LIN {X 0,Y 479.936,Z 1149.126,A -85,B 0,C 180,E1 22945.1,E2 22945.1} C_VEL
LIN {X 0,Y 479.98,Z 1146.25,A -85,B 0,C 180,E1 22942.699,E2 22942.699} C_VEL
LIN {X 0,Y 480.18,Z 1141.26,A -85,B 0,C 180,E1 22939.805,E2 22939.805} C_VEL
LIN {X 0,Y 480.58,Z 1135.396,A -85,B 0,C 180,E1 22937.259,E2 22937.259} C_VEL
LIN {X 0,Y 481.324,Z 1127.79,A -85,B 0,C 180,E1 22934.559,E2 22934.559} C_VEL
LIN {X 0,Y 482.53,Z 1118.085,A -85,B 0,C 180,E1 22931.766,E2 22931.766} C_VEL
LIN {X 0,Y 484.044,Z 1108.078,A -85,B 0,C 180,E1 22929.315,E2 22929.315} C_VEL
LIN {X 0,Y 486.397,Z 1094.541,A -85,B 0,C 180,E1 22926.496,E2 22926.496} C_VEL
LIN {X 0,Y 488.884,Z 1081.566,A -85,B 0,C 180,E1 22924.174,E2 22924.174} C_VEL
LIN {X 0,Y 492.333,Z 1064.667,A -85,B 0,C 180,E1 22921.569,E2 22921.569} C_VEL
LIN {X 0,Y 495.487,Z 1049.693,A -85,B 0,C 180,E1 22919.568,E2 22919.568} C_VEL
LIN {X 0,Y 499.695,Z 1030.069,A -85,B 0,C 180,E1 22917.298,E2 22917.298} C_VEL
LIN {X 0,Y 503.179,Z 1013.547,A -85,B 0,C 180,E1 22915.643,E2 22915.643} C_VEL
LIN {X 0,Y 507.434,Z 992.772,A -85,B 0,C 180,E1 22913.831,E2 22913.831} C_VEL
LIN {X 0,Y 511.179,Z 973.376,A -85,B 0,C 180,E1 22912.39,E2 22912.39} C_VEL
LIN {X 0,Y 515.064,Z 952.143,A -85,B 0,C 180,E1 22911.025,E2 22911.025} C_VEL
LIN {X 0,Y 518.682,Z 929.949,A -85,B 0,C 180,E1 22909.847,E2 22909.847} C_VEL
LIN {X 0,Y 521.763,Z 908.924,A -85,B 0,C 180,E1 22908.904,E2 22908.904} C_VEL
LIN {X 0,Y 524.789,Z 884.711,A -85,B 0,C 180,E1 22908.037,E2 22908.037} C_VEL
LIN {X 0,Y 526.942,Z 864.005,A -85,B 0,C 180,E1 22907.454,E2 22907.454} C_VEL
LIN {X 0,Y 528.934,Z 837.954,A -85,B 0,C 180,E1 22906.906,E2 22906.906} C_VEL
LIN {X 0,Y 532.506,Z 738.203,A -85,B 0,C 180,E1 22905.426,E2 22905.426} C_VEL
LIN {X 0,Y 540.091,Z 525.584,A -85,B 0,C 180,E1 22902.307,E2 22902.307} C_VEL
LIN {X 0,Y 527.108,Z 502.779,A -85,B 0,C 180,E1 22900.359,E2 22900.359} C_VEL
LIN {X 0,Y 515.721,Z 484.407,A -85,B 0,C 180,E1 22898.542,E2 22898.542} C_VEL
LIN {X 0,Y 504.612,Z 467.762,A -85,B 0,C 180,E1 22896.65,E2 22896.65} C_VEL
LIN {X 0,Y 495.161,Z 454.362,A -85,B 0,C 180,E1 22894.923,E2 22894.923} C_VEL
LIN {X 0,Y 490.761,Z 448.32,A -85,B 0,C 180,E1 22894.076,E2 22894.076} C_VEL
LIN {X 0,Y 486.838,Z 442.815,A -85,B 0,C 180,E1 22893.256,E2 22893.256} C_VEL
LIN {X 0,Y 485.319,Z 439.73,A -85,B 0,C 180,E1 22892.578,E2 22892.578} C_VEL
LIN {X 0,Y 483.506,Z 435.88,A -85,B 0,C 180,E1 22891.687,E2 22891.687} C_VEL
LIN {X 0,Y 482.074,Z 432.296,A -85,B 0,C 180,E1 22890.818,E2 22890.818} C_VEL
LIN {X 0,Y 482.051,Z 432.169,A -85,B 0,C 180,E1 22887.151,E2 22887.151} C_VEL
LIN {X 0,Y 482.046,Z 432.145,A -85,B 0,C 180,E1 22883.469,E2 22883.469} C_VEL
LIN {X 0,Y 482.039,Z 432.153,A -85,B 0,C 180,E1 22879.888,E2 22879.888} C_VEL
LIN {X 0,Y 482.05,Z 432.185,A -85,B 0,C 180,E1 22876.262,E2 22876.262} C_VEL
LIN {X 0,Y 482.037,Z 432.161,A -85,B 0,C 180,E1 22872.702,E2 22872.702} C_VEL
LIN {X 0,Y 482.034,Z 432.144,A -85,B 0,C 180,E1 22869.07,E2 22869.07} C_VEL
LIN {X 0,Y 482.052,Z 432.184,A -85,B 0,C 180,E1 22865.595,E2 22865.595} C_VEL
LIN {X 0,Y 482.048,Z 432.155,A -85,B 0,C 180,E1 22861.902,E2 22861.902} C_VEL
LIN {X 0,Y 482.023,Z 432.153,A -85,B 0,C 180,E1 22858.455,E2 22858.455} C_VEL
LIN {X 0,Y 482.023,Z 432.189,A -85,B 0,C 180,E1 22854.763,E2 22854.763} C_VEL
LIN {X 0,Y 482.046,Z 432.143,A -85,B 0,C 180,E1 22851.291,E2 22851.291} C_VEL
LIN {X 0,Y 482.044,Z 432.158,A -85,B 0,C 180,E1 22847.684,E2 22847.684} C_VEL
LIN {X 0,Y 482.01,Z 432.184,A -85,B 0,C 180,E1 22844.232,E2 22844.232} C_VEL
LIN {X 0,Y 482.005,Z 432.151,A -85,B 0,C 180,E1 22840.615,E2 22840.615} C_VEL
LIN {X 0,Y 482.051,Z 432.155,A -85,B 0,C 180,E1 22837.177,E2 22837.177} C_VEL
LIN {X 0,Y 482.022,Z 432.188,A -85,B 0,C 180,E1 22833.646,E2 22833.646} C_VEL
LIN {X 0,Y 481.988,Z 432.17,A -85,B 0,C 180,E1 22830.14,E2 22830.14} C_VEL
LIN {X 0,Y 482.003,Z 432.159,A -85,B 0,C 180,E1 22826.651,E2 22826.651} C_VEL
LIN {X 0,Y 482.017,Z 432.353,A -85,B 0,C 180,E1 22824.491,E2 22824.491} C_VEL
LIN {X 0,Y 482.37,Z 433.835,A -85,B 0,C 180,E1 22824.192,E2 22824.192} C_VEL
LIN {X 0,Y 484.285,Z 436.852,A -85,B 0,C 180,E1 22823.771,E2 22823.771} C_VEL
LIN {X 0,Y 486.647,Z 438.772,A -85,B 0,C 180,E1 22823.317,E2 22823.317} C_VEL
LIN {X 0,Y 489.004,Z 442.512,A -85,B 0,C 180,E1 22822.827,E2 22822.827} C_VEL
LIN {X 0,Y 491.314,Z 444.857,A -85,B 0,C 180,E1 22822.39,E2 22822.39} C_VEL
LIN {X 0,Y 494.506,Z 449.067,A -85,B 0,C 180,E1 22821.776,E2 22821.776} C_VEL
LIN {X 0,Y 496.224,Z 451.276,A -85,B 0,C 180,E1 22821.454,E2 22821.454} C_VEL
LIN {X 0,Y 503.923,Z 461.08,A -85,B 0,C 180,E1 22820.067,E2 22820.067} C_VEL
LIN {X 0,Y 515.356,Z 476.674,A -85,B 0,C 180,E1 22818.131,E2 22818.131} C_VEL
LIN {X 0,Y 527.952,Z 494.875,A -85,B 0,C 180,E1 22816.156,E2 22816.156} C_VEL
LIN {X 0,Y 540.315,Z 514.018,A -85,B 0,C 180,E1 22814.349,E2 22814.349} C_VEL
LIN {X 0,Y 531.611,Z 754.844,A -85,B 0,C 180,E1 22810.823,E2 22810.823} C_VEL
LIN {X 0,Y 529.419,Z 812.429,A -85,B 0,C 180,E1 22809.954,E2 22809.954} C_VEL
LIN {X 0,Y 527.614,Z 836.833,A -85,B 0,C 180,E1 22809.41,E2 22809.41} C_VEL
LIN {X 0,Y 525.485,Z 858.718,A -85,B 0,C 180,E1 22808.766,E2 22808.766} C_VEL
LIN {X 0,Y 522.555,Z 882.977,A -85,B 0,C 180,E1 22807.847,E2 22807.847} C_VEL
LIN {X 0,Y 519.79,Z 902.352,A -85,B 0,C 180,E1 22806.952,E2 22806.952} C_VEL
LIN {X 0,Y 516.232,Z 924.536,A -85,B 0,C 180,E1 22805.738,E2 22805.738} C_VEL
LIN {X 0,Y 512.66,Z 944.242,A -85,B 0,C 180,E1 22804.445,E2 22804.445} C_VEL
LIN {X 0,Y 509.031,Z 962.981,A -85,B 0,C 180,E1 22803.031,E2 22803.031} C_VEL
LIN {X 0,Y 504.72,Z 983.574,A -85,B 0,C 180,E1 22801.214,E2 22801.214} C_VEL
LIN {X 0,Y 501.128,Z 1000.134,A -85,B 0,C 180,E1 22799.527,E2 22799.527} C_VEL
LIN {X 0,Y 499.238,Z 1008.711,A -85,B 0,C 180,E1 22798.556,E2 22798.556} C_VEL
LIN {X 0,Y 497.144,Z 1014.273,A -85,B 0,C 180,E1 22797.965,E2 22797.965} C_VEL
LIN {X 0,Y 488.33,Z 1028.661,A -85,B 0,C 180,E1 22796.469,E2 22796.469} C_VEL
LIN {X 0,Y 486.663,Z 1032.843,A -85,B 0,C 180,E1 22795.904,E2 22795.904} C_VEL
LIN {X 0,Y 483.204,Z 1047.996,A -85,B 0,C 180,E1 22793.539,E2 22793.539} C_VEL
LIN {X 0,Y 480.254,Z 1061.231,A -85,B 0,C 180,E1 22791.112,E2 22791.112} C_VEL
LIN {X 0,Y 477.712,Z 1073.52,A -85,B 0,C 180,E1 22788.527,E2 22788.527} C_VEL
LIN {X 0,Y 475.693,Z 1084.165,A -85,B 0,C 180,E1 22785.858,E2 22785.858} C_VEL
LIN {X 0,Y 474.325,Z 1092.525,A -85,B 0,C 180,E1 22783.408,E2 22783.408} C_VEL
LIN {X 0,Y 473.141,Z 1101.135,A -85,B 0,C 180,E1 22780.348,E2 22780.348} C_VEL
LIN {X 0,Y 472.538,Z 1106.877,A -85,B 0,C 180,E1 22777.783,E2 22777.783} C_VEL
LIN {X 0,Y 472.182,Z 1111.811,A -85,B 0,C 180,E1 22774.981,E2 22774.981} C_VEL
LIN {X 0,Y 472.022,Z 1115.222,A -85,B 0,C 180,E1 22772.064,E2 22772.064} C_VEL
LIN {X 0,Y 471.975,Z 1117.08,A -85,B 0,C 180,E1 22769.42,E2 22769.42} C_VEL
LIN {X 0,Y 471.949,Z 1117.65,A -85,B 0,C 180,E1 22766.477,E2 22766.477} C_VEL
LIN {X 0,Y 471.985,Z 1116.842,A -85,B 0,C 180,E1 22763.92,E2 22763.92} C_VEL
LIN {X 0,Y 472.055,Z 1114.793,A -85,B 0,C 180,E1 22761.228,E2 22761.228} C_VEL
LIN {X 0,Y 472.266,Z 1110.779,A -85,B 0,C 180,E1 22758.149,E2 22758.149} C_VEL
LIN {X 0,Y 472.687,Z 1106.041,A -85,B 0,C 180,E1 22755.546,E2 22755.546} C_VEL
LIN {X 0,Y 473.537,Z 1099.04,A -85,B 0,C 180,E1 22752.552,E2 22752.552} C_VEL
LIN {X 0,Y 474.692,Z 1091.317,A -85,B 0,C 180,E1 22749.919,E2 22749.919} C_VEL
LIN {X 0,Y 476.475,Z 1081.561,A -85,B 0,C 180,E1 22747.11,E2 22747.11} C_VEL
LIN {X 0,Y 478.802,Z 1070.113,A -85,B 0,C 180,E1 22744.387,E2 22744.387} C_VEL
LIN {X 0,Y 481.716,Z 1057.311,A -85,B 0,C 180,E1 22741.754,E2 22741.754} C_VEL
LIN {X 0,Y 485.097,Z 1042.937,A -85,B 0,C 180,E1 22739.257,E2 22739.257} C_VEL
LIN {X 0,Y 488.946,Z 1027.419,A -85,B 0,C 180,E1 22736.906,E2 22736.906} C_VEL
LIN {X 0,Y 493.024,Z 1010.801,A -85,B 0,C 180,E1 22734.761,E2 22734.761} C_VEL
LIN {X 0,Y 496.931,Z 994.799,A -85,B 0,C 180,E1 22732.946,E2 22732.946} C_VEL
LIN {X 0,Y 501.49,Z 975.341,A -85,B 0,C 180,E1 22731.042,E2 22731.042} C_VEL
LIN {X 0,Y 505.451,Z 957.608,A -85,B 0,C 180,E1 22729.544,E2 22729.544} C_VEL
LIN {X 0,Y 510.033,Z 935.666,A -85,B 0,C 180,E1 22727.954,E2 22727.954} C_VEL
LIN {X 0,Y 513.708,Z 916.026,A -85,B 0,C 180,E1 22726.753,E2 22726.753} C_VEL
LIN {X 0,Y 517.485,Z 894.109,A -85,B 0,C 180,E1 22725.616,E2 22725.616} C_VEL
LIN {X 0,Y 520.64,Z 871.877,A -85,B 0,C 180,E1 22724.678,E2 22724.678} C_VEL
LIN {X 0,Y 523.211,Z 850.767,A -85,B 0,C 180,E1 22723.951,E2 22723.951} C_VEL
LIN {X 0,Y 525.614,Z 825.467,A -85,B 0,C 180,E1 22723.286,E2 22723.286} C_VEL
LIN {X 0,Y 527.005,Z 803.925,A -85,B 0,C 180,E1 22722.873,E2 22722.873} C_VEL
LIN {X 0,Y 537.124,Z 553.916,A -85,B 0,C 180,E1 22719.149,E2 22719.149} C_VEL
LIN {X 0,Y 538.478,Z 519.428,A -85,B 0,C 180,E1 22718.621,E2 22718.621} C_VEL
LIN {X 0,Y 526.57,Z 501.373,A -85,B 0,C 180,E1 22716.67,E2 22716.67} C_VEL
LIN {X 0,Y 513.397,Z 482.898,A -85,B 0,C 180,E1 22714.328,E2 22714.328} C_VEL
LIN {X 0,Y 502.204,Z 468.261,A -85,B 0,C 180,E1 22712.147,E2 22712.147} C_VEL
LIN {X 0,Y 496.887,Z 461.776,A -85,B 0,C 180,E1 22711.041,E2 22711.041} C_VEL
LIN {X 0,Y 492.914,Z 456.709,A -85,B 0,C 180,E1 22710.17,E2 22710.17} C_VEL
LIN {X 0,Y 489.386,Z 452.141,A -85,B 0,C 180,E1 22709.364,E2 22709.364} C_VEL
LIN {X 0,Y 485.532,Z 448.038,A -85,B 0,C 180,E1 22708.473,E2 22708.473} C_VEL
LIN {X 0,Y 484.051,Z 445.687,A -85,B 0,C 180,E1 22708.098,E2 22708.098} C_VEL
LIN {X 0,Y 480.94,Z 442.93,A -85,B 0,C 180,E1 22707.353,E2 22707.353} C_VEL
LIN {X 0,Y 478.923,Z 439.552,A -85,B 0,C 180,E1 22706.806,E2 22706.806} C_VEL
LIN {X 0,Y 475.792,Z 437.238,A -85,B 0,C 180,E1 22706.021,E2 22706.021} C_VEL
LIN {X 0,Y 474.203,Z 433.97,A -85,B 0,C 180,E1 22705.477,E2 22705.477} C_VEL
LIN {X 0,Y 474.091,Z 433.21,A -85,B 0,C 180,E1 22705.083,E2 22705.083} C_VEL
LIN {X 0,Y 474.059,Z 433.17,A -85,B 0,C 180,E1 22701.661,E2 22701.661} C_VEL
LIN {X 0,Y 474.081,Z 433.179,A -85,B 0,C 180,E1 22698.062,E2 22698.062} C_VEL
LIN {X 0,Y 474.123,Z 433.153,A -85,B 0,C 180,E1 22694.533,E2 22694.533} C_VEL
LIN {X 0,Y 474.093,Z 433.142,A -85,B 0,C 180,E1 22690.942,E2 22690.942} C_VEL
LIN {X 0,Y 474.072,Z 433.146,A -85,B 0,C 180,E1 22687.392,E2 22687.392} C_VEL
LIN {X 0,Y 474.087,Z 433.165,A -85,B 0,C 180,E1 22683.749,E2 22683.749} C_VEL
LIN {X 0,Y 474.121,Z 433.16,A -85,B 0,C 180,E1 22680.121,E2 22680.121} C_VEL
LIN {X 0,Y 474.106,Z 433.137,A -85,B 0,C 180,E1 22676.494,E2 22676.494} C_VEL
LIN {X 0,Y 474.1,Z 433.137,A -85,B 0,C 180,E1 22672.852,E2 22672.852} C_VEL
LIN {X 0,Y 474.095,Z 433.156,A -85,B 0,C 180,E1 22669.181,E2 22669.181} C_VEL
LIN {X 0,Y 474.108,Z 433.175,A -85,B 0,C 180,E1 22665.465,E2 22665.465} C_VEL
LIN {X 0,Y 474.109,Z 433.157,A -85,B 0,C 180,E1 22661.812,E2 22661.812} C_VEL
LIN {X 0,Y 474.095,Z 433.122,A -85,B 0,C 180,E1 22658.123,E2 22658.123} C_VEL
LIN {X 0,Y 474.105,Z 433.14,A -85,B 0,C 180,E1 22654.51,E2 22654.51} C_VEL
LIN {X 0,Y 474.169,Z 433.53,A -85,B 0,C 180,E1 22653.136,E2 22653.136} C_VEL
LIN {X 0,Y 475.766,Z 437.121,A -85,B 0,C 180,E1 22652.052,E2 22652.052} C_VEL
LIN {X 0,Y 476.842,Z 439.144,A -85,B 0,C 180,E1 22651.439,E2 22651.439} C_VEL
LIN {X 0,Y 478.321,Z 441.84,A -85,B 0,C 180,E1 22650.749,E2 22650.749} C_VEL
LIN {X 0,Y 480.674,Z 444.989,A -85,B 0,C 180,E1 22650.119,E2 22650.119} C_VEL
LIN {X 0,Y 484.461,Z 449.557,A -85,B 0,C 180,E1 22649.178,E2 22649.178} C_VEL
LIN {X 0,Y 493.093,Z 461.044,A -85,B 0,C 180,E1 22647.15,E2 22647.15} C_VEL
LIN {X 0,Y 496.711,Z 465.928,A -85,B 0,C 180,E1 22646.352,E2 22646.352} C_VEL
LIN {X 0,Y 505.532,Z 478.146,A -85,B 0,C 180,E1 22644.513,E2 22644.513} C_VEL
LIN {X 0,Y 517.369,Z 495.765,A -85,B 0,C 180,E1 22642.236,E2 22642.236} C_VEL
LIN {X 0,Y 529.249,Z 514.827,A -85,B 0,C 180,E1 22640.138,E2 22640.138} C_VEL
LIN {X 0,Y 538.374,Z 530.866,A -85,B 0,C 180,E1 22638.624,E2 22638.624} C_VEL
LIN {X 0,Y 529.453,Z 752.304,A -85,B 0,C 180,E1 22635.324,E2 22635.324} C_VEL
LIN {X 0,Y 525.979,Z 837.792,A -85,B 0,C 180,E1 22634.032,E2 22634.032} C_VEL
LIN {X 0,Y 523.839,Z 863.39,A -85,B 0,C 180,E1 22633.489,E2 22633.489} C_VEL
LIN {X 0,Y 521.554,Z 883.538,A -85,B 0,C 180,E1 22632.923,E2 22632.923} C_VEL
LIN {X 0,Y 518.464,Z 906.572,A -85,B 0,C 180,E1 22632.109,E2 22632.109} C_VEL
LIN {X 0,Y 515.038,Z 927.934,A -85,B 0,C 180,E1 22631.158,E2 22631.158} C_VEL
LIN {X 0,Y 511.484,Z 947.966,A -85,B 0,C 180,E1 22630.101,E2 22630.101} C_VEL
LIN {X 0,Y 506.92,Z 971.138,A -85,B 0,C 180,E1 22628.638,E2 22628.638} C_VEL
LIN {X 0,Y 502.967,Z 989.767,A -85,B 0,C 180,E1 22627.254,E2 22627.254} C_VEL
LIN {X 0,Y 498.144,Z 1011.239,A -85,B 0,C 180,E1 22625.394,E2 22625.394} C_VEL
LIN {X 0,Y 494.168,Z 1028.309,A -85,B 0,C 180,E1 22623.67,E2 22623.67} C_VEL
LIN {X 0,Y 490.033,Z 1046.043,A -85,B 0,C 180,E1 22621.628,E2 22621.628} C_VEL
LIN {X 0,Y 486.163,Z 1062.323,A -85,B 0,C 180,E1 22619.443,E2 22619.443} C_VEL
LIN {X 0,Y 482.714,Z 1077.589,A -85,B 0,C 180,E1 22617.111,E2 22617.111} C_VEL
LIN {X 0,Y 479.55,Z 1092.099,A -85,B 0,C 180,E1 22614.515,E2 22614.515} C_VEL
LIN {X 0,Y 477.183,Z 1104.197,A -85,B 0,C 180,E1 22612.029,E2 22612.029} C_VEL
LIN {X 0,Y 475.106,Z 1116.023,A -85,B 0,C 180,E1 22609.166,E2 22609.166} C_VEL
LIN {X 0,Y 473.768,Z 1125.193,A -85,B 0,C 180,E1 22606.554,E2 22606.554} C_VEL
LIN {X 0,Y 472.752,Z 1134.133,A -85,B 0,C 180,E1 22603.453,E2 22603.453} C_VEL
LIN {X 0,Y 472.266,Z 1140.124,A -85,B 0,C 180,E1 22600.861,E2 22600.861} C_VEL
LIN {X 0,Y 471.998,Z 1145.405,A -85,B 0,C 180,E1 22597.915,E2 22597.915} C_VEL
LIN {X 0,Y 471.932,Z 1148.649,A -85,B 0,C 180,E1 22595.252,E2 22595.252} C_VEL
LIN {X 0,Y 471.932,Z 1150.44,A -85,B 0,C 180,E1 22592.915,E2 22592.915} C_VEL
LIN {X 0,Y 471.949,Z 1151.281,A -85,B 0,C 180,E1 22590.243,E2 22590.243} C_VEL
LIN {X 0,Y 471.94,Z 1150.604,A -85,B 0,C 180,E1 22587.45,E2 22587.45} C_VEL
LIN {X 0,Y 471.937,Z 1148.827,A -85,B 0,C 180,E1 22585.017,E2 22585.017} C_VEL
LIN {X 0,Y 471.98,Z 1145.943,A -85,B 0,C 180,E1 22582.575,E2 22582.575} C_VEL
LIN {X 0,Y 472.199,Z 1140.94,A -85,B 0,C 180,E1 22579.631,E2 22579.631} C_VEL
LIN {X 0,Y 472.625,Z 1135.067,A -85,B 0,C 180,E1 22577.041,E2 22577.041} C_VEL
LIN {X 0,Y 473.411,Z 1127.509,A -85,B 0,C 180,E1 22574.315,E2 22574.315} C_VEL
LIN {X 0,Y 474.701,Z 1117.728,A -85,B 0,C 180,E1 22571.454,E2 22571.454} C_VEL
LIN {X 0,Y 476.296,Z 1107.71,A -85,B 0,C 180,E1 22568.962,E2 22568.962} C_VEL
LIN {X 0,Y 478.782,Z 1094.151,A -85,B 0,C 180,E1 22566.099,E2 22566.099} C_VEL
LIN {X 0,Y 481.301,Z 1081.658,A -85,B 0,C 180,E1 22563.828,E2 22563.828} C_VEL
LIN {X 0,Y 484.946,Z 1064.601,A -85,B 0,C 180,E1 22561.153,E2 22561.153} C_VEL
LIN {X 0,Y 488.302,Z 1049.388,A -85,B 0,C 180,E1 22559.091,E2 22559.091} C_VEL
LIN {X 0,Y 492.724,Z 1029.594,A -85,B 0,C 180,E1 22556.776,E2 22556.776} C_VEL
LIN {X 0,Y 496.453,Z 1012.59,A -85,B 0,C 180,E1 22555.058,E2 22555.058} C_VEL
LIN {X 0,Y 501.127,Z 990.544,A -85,B 0,C 180,E1 22553.141,E2 22553.141} C_VEL
LIN {X 0,Y 504.863,Z 971.911,A -85,B 0,C 180,E1 22551.756,E2 22551.756} C_VEL
LIN {X 0,Y 509.062,Z 949.487,A -85,B 0,C 180,E1 22550.33,E2 22550.33} C_VEL
LIN {X 0,Y 512.46,Z 929.277,A -85,B 0,C 180,E1 22549.257,E2 22549.257} C_VEL
LIN {X 0,Y 515.769,Z 907.446,A -85,B 0,C 180,E1 22548.278,E2 22548.278} C_VEL
LIN {X 0,Y 518.777,Z 883.834,A -85,B 0,C 180,E1 22547.437,E2 22547.437} C_VEL
LIN {X 0,Y 520.974,Z 863.298,A -85,B 0,C 180,E1 22546.859,E2 22546.859} C_VEL
LIN {X 0,Y 523.033,Z 836.601,A -85,B 0,C 180,E1 22546.3,E2 22546.3} C_VEL
LIN {X 0,Y 530.859,Z 624.102,A -85,B 0,C 180,E1 22543.147,E2 22543.147} C_VEL
LIN {X 0,Y 534.336,Z 528.71,A -85,B 0,C 180,E1 22541.719,E2 22541.719} C_VEL
LIN {X 0,Y 521.84,Z 506.736,A -85,B 0,C 180,E1 22539.79,E2 22539.79} C_VEL
LIN {X 0,Y 509.772,Z 487.18,A -85,B 0,C 180,E1 22537.803,E2 22537.803} C_VEL
LIN {X 0,Y 497.334,Z 468.611,A -85,B 0,C 180,E1 22535.594,E2 22535.594} C_VEL
LIN {X 0,Y 487.735,Z 455.202,A -85,B 0,C 180,E1 22533.75,E2 22533.75} C_VEL
LIN {X 0,Y 481.103,Z 446.349,A -85,B 0,C 180,E1 22532.391,E2 22532.391} C_VEL
LIN {X 0,Y 478.14,Z 441.839,A -85,B 0,C 180,E1 22531.661,E2 22531.661} C_VEL
LIN {X 0,Y 475.595,Z 436.916,A -85,B 0,C 180,E1 22530.443,E2 22530.443} C_VEL
LIN {X 0,Y 474.129,Z 433.295,A -85,B 0,C 180,E1 22529.5,E2 22529.5} C_VEL
LIN {X 0,Y 474.098,Z 433.161,A -85,B 0,C 180,E1 22525.885,E2 22525.885} C_VEL
LIN {X 0,Y 474.102,Z 433.162,A -85,B 0,C 180,E1 22522.18,E2 22522.18} C_VEL
LIN {X 0,Y 474.106,Z 433.137,A -85,B 0,C 180,E1 22518.57,E2 22518.57} C_VEL
LIN {X 0,Y 474.1,Z 433.139,A -85,B 0,C 180,E1 22514.91,E2 22514.91} C_VEL
LIN {X 0,Y 474.108,Z 433.175,A -85,B 0,C 180,E1 22511.279,E2 22511.279} C_VEL
LIN {X 0,Y 474.11,Z 433.139,A -85,B 0,C 180,E1 22507.595,E2 22507.595} C_VEL
LIN {X 0,Y 474.105,Z 433.136,A -85,B 0,C 180,E1 22503.991,E2 22503.991} C_VEL
LIN {X 0,Y 474.092,Z 433.176,A -85,B 0,C 180,E1 22500.363,E2 22500.363} C_VEL
LIN {X 0,Y 474.081,Z 433.136,A -85,B 0,C 180,E1 22496.735,E2 22496.735} C_VEL
LIN {X 0,Y 474.11,Z 433.144,A -85,B 0,C 180,E1 22493.217,E2 22493.217} C_VEL
LIN {X 0,Y 474.113,Z 433.169,A -85,B 0,C 180,E1 22489.55,E2 22489.55} C_VEL
LIN {X 0,Y 474.081,Z 433.133,A -85,B 0,C 180,E1 22485.963,E2 22485.963} C_VEL
LIN {X 0,Y 474.067,Z 433.155,A -85,B 0,C 180,E1 22482.43,E2 22482.43} C_VEL
LIN {X 0,Y 474.084,Z 433.172,A -85,B 0,C 180,E1 22478.859,E2 22478.859} C_VEL
LIN {X 0,Y 474.104,Z 433.136,A -85,B 0,C 180,E1 22475.366,E2 22475.366} C_VEL
LIN {X 0,Y 474.064,Z 433.143,A -85,B 0,C 180,E1 22471.806,E2 22471.806} C_VEL
LIN {X 0,Y 474.048,Z 433.159,A -85,B 0,C 180,E1 22468.216,E2 22468.216} C_VEL
LIN {X 0,Y 474.06,Z 433.271,A -85,B 0,C 180,E1 22465.944,E2 22465.944} C_VEL
LIN {X 0,Y 474.423,Z 434.745,A -85,B 0,C 180,E1 22465.624,E2 22465.624} C_VEL
LIN {X 0,Y 476.306,Z 437.77,A -85,B 0,C 180,E1 22465.18,E2 22465.18} C_VEL
LIN {X 0,Y 478.828,Z 439.895,A -85,B 0,C 180,E1 22464.659,E2 22464.659} C_VEL
LIN {X 0,Y 481.264,Z 443.655,A -85,B 0,C 180,E1 22464.123,E2 22464.123} C_VEL
LIN {X 0,Y 483.6,Z 445.904,A -85,B 0,C 180,E1 22463.656,E2 22463.656} C_VEL
LIN {X 0,Y 486.679,Z 450.083,A -85,B 0,C 180,E1 22463.025,E2 22463.025} C_VEL
LIN {X 0,Y 488.487,Z 452.236,A -85,B 0,C 180,E1 22462.67,E2 22462.67} C_VEL
LIN {X 0,Y 493.304,Z 458.45,A -85,B 0,C 180,E1 22461.74,E2 22461.74} C_VEL
LIN {X 0,Y 500.474,Z 467.61,A -85,B 0,C 180,E1 22460.426,E2 22460.426} C_VEL
LIN {X 0,Y 511.731,Z 483.101,A -85,B 0,C 180,E1 22458.48,E2 22458.48} C_VEL
LIN {X 0,Y 524.073,Z 501.11,A -85,B 0,C 180,E1 22456.505,E2 22456.505} C_VEL
LIN {X 0,Y 534.671,Z 517.793,A -85,B 0,C 180,E1 22454.915,E2 22454.915} C_VEL
LIN {X 0,Y 525.544,Z 760.909,A -85,B 0,C 180,E1 22451.329,E2 22451.329} C_VEL
LIN {X 0,Y 523.446,Z 813.486,A -85,B 0,C 180,E1 22450.524,E2 22450.524} C_VEL
LIN {X 0,Y 521.571,Z 837.655,A -85,B 0,C 180,E1 22449.976,E2 22449.976} C_VEL
LIN {X 0,Y 519.314,Z 860.093,A -85,B 0,C 180,E1 22449.306,E2 22449.306} C_VEL
LIN {X 0,Y 516.425,Z 883.033,A -85,B 0,C 180,E1 22448.427,E2 22448.427} C_VEL
LIN {X 0,Y 513.451,Z 903.213,A -85,B 0,C 180,E1 22447.486,E2 22447.486} C_VEL
LIN {X 0,Y 509.588,Z 926.256,A -85,B 0,C 180,E1 22446.2,E2 22446.2} C_VEL
LIN {X 0,Y 505.899,Z 945.877,A -85,B 0,C 180,E1 22444.891,E2 22444.891} C_VEL
LIN {X 0,Y 501.75,Z 966.474,A -85,B 0,C 180,E1 22443.3,E2 22443.3} C_VEL
LIN {X 0,Y 497.537,Z 985.58,A -85,B 0,C 180,E1 22441.558,E2 22441.558} C_VEL
LIN {X 0,Y 493.351,Z 1004.247,A -85,B 0,C 180,E1 22439.603,E2 22439.603} C_VEL
LIN {X 0,Y 489.356,Z 1021.307,A -85,B 0,C 180,E1 22437.502,E2 22437.502} C_VEL
LIN {X 0,Y 486.663,Z 1032.843,A -85,B 0,C 180,E1 22435.904,E2 22435.904} C_VEL
LIN {X 0,Y 484.627,Z 1037.843,A -85,B 0,C 180,E1 22435.234,E2 22435.234} C_VEL
LIN {X 0,Y 476.305,Z 1049.996,A -85,B 0,C 180,E1 22433.6,E2 22433.6} C_VEL
LIN {X 0,Y 474.375,Z 1054.367,A -85,B 0,C 180,E1 22432.87,E2 22432.87} C_VEL
LIN {X 0,Y 471.109,Z 1068.831,A -85,B 0,C 180,E1 22429.981,E2 22429.981} C_VEL
LIN {X 0,Y 468.907,Z 1079.415,A -85,B 0,C 180,E1 22427.498,E2 22427.498} C_VEL
LIN {X 0,Y 466.861,Z 1090.562,A -85,B 0,C 180,E1 22424.385,E2 22424.385} C_VEL
LIN {X 0,Y 465.647,Z 1098.464,A -85,B 0,C 180,E1 22421.712,E2 22421.712} C_VEL
LIN {X 0,Y 464.717,Z 1105.998,A -85,B 0,C 180,E1 22418.538,E2 22418.538} C_VEL
LIN {X 0,Y 464.28,Z 1110.751,A -85,B 0,C 180,E1 22415.934,E2 22415.934} C_VEL
LIN {X 0,Y 464.063,Z 1114.639,A -85,B 0,C 180,E1 22413.088,E2 22413.088} C_VEL
LIN {X 0,Y 464.005,Z 1116.998,A -85,B 0,C 180,E1 22410.123,E2 22410.123} C_VEL
LIN {X 0,Y 463.958,Z 1117.893,A -85,B 0,C 180,E1 22407.53,E2 22407.53} C_VEL
LIN {X 0,Y 463.979,Z 1117.439,A -85,B 0,C 180,E1 22404.435,E2 22404.435} C_VEL
LIN {X 0,Y 464.047,Z 1115.6,A -85,B 0,C 180,E1 22401.699,E2 22401.699} C_VEL
LIN {X 0,Y 464.22,Z 1112.369,A -85,B 0,C 180,E1 22398.822,E2 22398.822} C_VEL
LIN {X 0,Y 464.655,Z 1107.257,A -85,B 0,C 180,E1 22395.799,E2 22395.799} C_VEL
LIN {X 0,Y 465.357,Z 1101.455,A -85,B 0,C 180,E1 22393.138,E2 22393.138} C_VEL
LIN {X 0,Y 466.722,Z 1092.696,A -85,B 0,C 180,E1 22389.954,E2 22389.954} C_VEL
LIN {X 0,Y 468.316,Z 1084.161,A -85,B 0,C 180,E1 22387.399,E2 22387.399} C_VEL
LIN {X 0,Y 470.925,Z 1071.955,A -85,B 0,C 180,E1 22384.333,E2 22384.333} C_VEL
LIN {X 0,Y 473.577,Z 1060.588,A -85,B 0,C 180,E1 22381.911,E2 22381.911} C_VEL
LIN {X 0,Y 477.265,Z 1045.788,A -85,B 0,C 180,E1 22379.201,E2 22379.201} C_VEL
LIN {X 0,Y 480.854,Z 1031.702,A -85,B 0,C 180,E1 22376.989,E2 22376.989} C_VEL
LIN {X 0,Y 485.368,Z 1014.37,A -85,B 0,C 180,E1 22374.628,E2 22374.628} C_VEL
LIN {X 0,Y 489.446,Z 998.29,A -85,B 0,C 180,E1 22372.746,E2 22372.746} C_VEL
LIN {X 0,Y 494.075,Z 979.746,A -85,B 0,C 180,E1 22370.845,E2 22370.845} C_VEL
LIN {X 0,Y 498.541,Z 960.464,A -85,B 0,C 180,E1 22369.168,E2 22369.168} C_VEL
LIN {X 0,Y 502.778,Z 941.198,A -85,B 0,C 180,E1 22367.715,E2 22367.715} C_VEL
LIN {X 0,Y 507.119,Z 919.301,A -85,B 0,C 180,E1 22366.32,E2 22366.32} C_VEL
LIN {X 0,Y 510.741,Z 899.097,A -85,B 0,C 180,E1 22365.238,E2 22365.238} C_VEL
LIN {X 0,Y 514.539,Z 874.389,A -85,B 0,C 180,E1 22364.147,E2 22364.147} C_VEL
LIN {X 0,Y 517.198,Z 853.451,A -85,B 0,C 180,E1 22363.407,E2 22363.407} C_VEL
LIN {X 0,Y 519.756,Z 828.599,A -85,B 0,C 180,E1 22362.725,E2 22362.725} C_VEL
LIN {X 0,Y 521.316,Z 805.933,A -85,B 0,C 180,E1 22362.277,E2 22362.277} C_VEL
LIN {X 0,Y 531.53,Z 563.128,A -85,B 0,C 180,E1 22358.631,E2 22358.631} C_VEL
LIN {X 0,Y 533.235,Z 523.387,A -85,B 0,C 180,E1 22358.03,E2 22358.03} C_VEL
LIN {X 0,Y 521.943,Z 506.222,A -85,B 0,C 180,E1 22356.126,E2 22356.126} C_VEL
LIN {X 0,Y 509.696,Z 488.932,A -85,B 0,C 180,E1 22353.892,E2 22353.892} C_VEL
LIN {X 0,Y 499.038,Z 474.875,A -85,B 0,C 180,E1 22351.766,E2 22351.766} C_VEL
LIN {X 0,Y 493.434,Z 467.961,A -85,B 0,C 180,E1 22350.572,E2 22350.572} C_VEL
LIN {X 0,Y 489.86,Z 463.368,A -85,B 0,C 180,E1 22349.77,E2 22349.77} C_VEL
LIN {X 0,Y 485.917,Z 458.419,A -85,B 0,C 180,E1 22348.852,E2 22348.852} C_VEL
LIN {X 0,Y 482.383,Z 454.261,A -85,B 0,C 180,E1 22348.002,E2 22348.002} C_VEL
LIN {X 0,Y 481.32,Z 452.783,A -85,B 0,C 180,E1 22347.732,E2 22347.732} C_VEL
LIN {X 0,Y 477.967,Z 449.361,A -85,B 0,C 180,E1 22346.897,E2 22346.897} C_VEL
LIN {X 0,Y 476.25,Z 446.767,A -85,B 0,C 180,E1 22346.43,E2 22346.43} C_VEL
LIN {X 0,Y 473.103,Z 443.984,A -85,B 0,C 180,E1 22345.608,E2 22345.608} C_VEL
LIN {X 0,Y 471.223,Z 440.672,A -85,B 0,C 180,E1 22345.045,E2 22345.045} C_VEL
LIN {X 0,Y 467.883,Z 438.226,A -85,B 0,C 180,E1 22344.124,E2 22344.124} C_VEL
LIN {X 0,Y 466.263,Z 434.951,A -85,B 0,C 180,E1 22343.508,E2 22343.508} C_VEL
LIN {X 0,Y 466.159,Z 434.177,A -85,B 0,C 180,E1 22342.978,E2 22342.978} C_VEL
LIN {X 0,Y 466.126,Z 434.139,A -85,B 0,C 180,E1 22339.42,E2 22339.42} C_VEL
LIN {X 0,Y 466.128,Z 434.133,A -85,B 0,C 180,E1 22335.809,E2 22335.809} C_VEL
LIN {X 0,Y 466.162,Z 434.134,A -85,B 0,C 180,E1 22332.26,E2 22332.26} C_VEL
LIN {X 0,Y 466.178,Z 434.155,A -85,B 0,C 180,E1 22328.587,E2 22328.587} C_VEL
LIN {X 0,Y 466.158,Z 434.156,A -85,B 0,C 180,E1 22324.922,E2 22324.922} C_VEL
LIN {X 0,Y 466.144,Z 434.129,A -85,B 0,C 180,E1 22321.229,E2 22321.229} C_VEL
LIN {X 0,Y 466.148,Z 434.123,A -85,B 0,C 180,E1 22317.541,E2 22317.541} C_VEL
LIN {X 0,Y 466.17,Z 434.138,A -85,B 0,C 180,E1 22313.843,E2 22313.843} C_VEL
LIN {X 0,Y 466.173,Z 434.162,A -85,B 0,C 180,E1 22310.12,E2 22310.12} C_VEL
LIN {X 0,Y 466.168,Z 434.143,A -85,B 0,C 180,E1 22306.353,E2 22306.353} C_VEL
LIN {X 0,Y 466.164,Z 434.13,A -85,B 0,C 180,E1 22302.782,E2 22302.782} C_VEL
LIN {X 0,Y 466.164,Z 434.115,A -85,B 0,C 180,E1 22299.142,E2 22299.142} C_VEL
LIN {X 0,Y 466.172,Z 434.16,A -85,B 0,C 180,E1 22295.546,E2 22295.546} C_VEL
LIN {X 0,Y 466.25,Z 434.646,A -85,B 0,C 180,E1 22294.873,E2 22294.873} C_VEL
LIN {X 0,Y 467.82,Z 438.088,A -85,B 0,C 180,E1 22293.741,E2 22293.741} C_VEL
LIN {X 0,Y 468.97,Z 440.146,A -85,B 0,C 180,E1 22293.059,E2 22293.059} C_VEL
LIN {X 0,Y 472.33,Z 444.518,A -85,B 0,C 180,E1 22292.037,E2 22292.037} C_VEL
LIN {X 0,Y 477.82,Z 451.575,A -85,B 0,C 180,E1 22290.543,E2 22290.543} C_VEL
LIN {X 0,Y 481.863,Z 456.649,A -85,B 0,C 180,E1 22289.512,E2 22289.512} C_VEL
LIN {X 0,Y 489.945,Z 467.466,A -85,B 0,C 180,E1 22287.573,E2 22287.573} C_VEL
LIN {X 0,Y 497.176,Z 477.385,A -85,B 0,C 180,E1 22285.968,E2 22285.968} C_VEL
LIN {X 0,Y 506.9,Z 491.496,A -85,B 0,C 180,E1 22283.962,E2 22283.962} C_VEL
LIN {X 0,Y 518.453,Z 509.357,A -85,B 0,C 180,E1 22281.768,E2 22281.768} C_VEL
LIN {X 0,Y 530.467,Z 529.55,A -85,B 0,C 180,E1 22279.666,E2 22279.666} C_VEL
LIN {X 0,Y 533.048,Z 534.482,A -85,B 0,C 180,E1 22279.227,E2 22279.227} C_VEL
LIN {X 0,Y 523.844,Z 754.793,A -85,B 0,C 180,E1 22275.921,E2 22275.921} C_VEL
LIN {X 0,Y 520.347,Z 837.619,A -85,B 0,C 180,E1 22274.659,E2 22274.659} C_VEL
LIN {X 0,Y 518.135,Z 863.216,A -85,B 0,C 180,E1 22274.112,E2 22274.112} C_VEL
LIN {X 0,Y 515.763,Z 883.49,A -85,B 0,C 180,E1 22273.54,E2 22273.54} C_VEL
LIN {X 0,Y 512.506,Z 906.844,A -85,B 0,C 180,E1 22272.707,E2 22272.707} C_VEL
LIN {X 0,Y 508.987,Z 928.03,A -85,B 0,C 180,E1 22271.756,E2 22271.756} C_VEL
LIN {X 0,Y 505.13,Z 949.022,A -85,B 0,C 180,E1 22270.636,E2 22270.636} C_VEL
LIN {X 0,Y 500.55,Z 971.289,A -85,B 0,C 180,E1 22269.208,E2 22269.208} C_VEL
LIN {X 0,Y 496.49,Z 989.723,A -85,B 0,C 180,E1 22267.824,E2 22267.824} C_VEL
LIN {X 0,Y 491.398,Z 1011.451,A -85,B 0,C 180,E1 22265.919,E2 22265.919} C_VEL
LIN {X 0,Y 487.193,Z 1028.757,A -85,B 0,C 180,E1 22264.147,E2 22264.147} C_VEL
LIN {X 0,Y 482.529,Z 1047.763,A -85,B 0,C 180,E1 22261.898,E2 22261.898} C_VEL
LIN {X 0,Y 478.762,Z 1063.016,A -85,B 0,C 180,E1 22259.806,E2 22259.806} C_VEL
LIN {X 0,Y 475,Z 1078.882,A -85,B 0,C 180,E1 22257.316,E2 22257.316} C_VEL
LIN {X 0,Y 471.88,Z 1092.545,A -85,B 0,C 180,E1 22254.806,E2 22254.806} C_VEL
LIN {X 0,Y 469.303,Z 1105.147,A -85,B 0,C 180,E1 22252.155,E2 22252.155} C_VEL
LIN {X 0,Y 467.237,Z 1116.263,A -85,B 0,C 180,E1 22249.372,E2 22249.372} C_VEL
LIN {X 0,Y 465.84,Z 1125.37,A -85,B 0,C 180,E1 22246.716,E2 22246.716} C_VEL
LIN {X 0,Y 464.81,Z 1133.884,A -85,B 0,C 180,E1 22243.688,E2 22243.688} C_VEL
LIN {X 0,Y 464.289,Z 1139.869,A -85,B 0,C 180,E1 22241.05,E2 22241.05} C_VEL
LIN {X 0,Y 464.007,Z 1145.138,A -85,B 0,C 180,E1 22238.052,E2 22238.052} C_VEL
LIN {X 0,Y 463.938,Z 1148.283,A -85,B 0,C 180,E1 22235.442,E2 22235.442} C_VEL
LIN {X 0,Y 463.939,Z 1150.093,A -85,B 0,C 180,E1 22233.089,E2 22233.089} C_VEL
LIN {X 0,Y 463.947,Z 1150.929,A -85,B 0,C 180,E1 22230.617,E2 22230.617} C_VEL
LIN {X 0,Y 463.953,Z 1150.449,A -85,B 0,C 180,E1 22227.653,E2 22227.653} C_VEL
LIN {X 0,Y 463.941,Z 1148.644,A -85,B 0,C 180,E1 22225.054,E2 22225.054} C_VEL
LIN {X 0,Y 463.983,Z 1145.965,A -85,B 0,C 180,E1 22222.695,E2 22222.695} C_VEL
LIN {X 0,Y 464.176,Z 1141.395,A -85,B 0,C 180,E1 22219.826,E2 22219.826} C_VEL
LIN {X 0,Y 464.647,Z 1135.047,A -85,B 0,C 180,E1 22216.941,E2 22216.941} C_VEL
LIN {X 0,Y 465.434,Z 1127.757,A -85,B 0,C 180,E1 22214.247,E2 22214.247} C_VEL
LIN {X 0,Y 466.841,Z 1117.646,A -85,B 0,C 180,E1 22211.207,E2 22211.207} C_VEL
LIN {X 0,Y 468.472,Z 1107.865,A -85,B 0,C 180,E1 22208.725,E2 22208.725} C_VEL
LIN {X 0,Y 471.064,Z 1094.407,A -85,B 0,C 180,E1 22205.816,E2 22205.816} C_VEL
LIN {X 0,Y 473.684,Z 1081.976,A -85,B 0,C 180,E1 22203.511,E2 22203.511} C_VEL
LIN {X 0,Y 477.103,Z 1066.757,A -85,B 0,C 180,E1 22201.045,E2 22201.045} C_VEL
LIN {X 0,Y 480.767,Z 1050.692,A -85,B 0,C 180,E1 22198.811,E2 22198.811} C_VEL
LIN {X 0,Y 484.923,Z 1033.073,A -85,B 0,C 180,E1 22196.666,E2 22196.666} C_VEL
LIN {X 0,Y 489.155,Z 1014.413,A -85,B 0,C 180,E1 22194.727,E2 22194.727} C_VEL
LIN {X 0,Y 493.504,Z 994.998,A -85,B 0,C 180,E1 22192.967,E2 22192.967} C_VEL
LIN {X 0,Y 497.899,Z 973.893,A -85,B 0,C 180,E1 22191.35,E2 22191.35} C_VEL
LIN {X 0,Y 502.052,Z 952.797,A -85,B 0,C 180,E1 22189.962,E2 22189.962} C_VEL
LIN {X 0,Y 505.914,Z 930.892,A -85,B 0,C 180,E1 22188.766,E2 22188.766} C_VEL
LIN {X 0,Y 508.983,Z 911.37,A -85,B 0,C 180,E1 22187.865,E2 22187.865} C_VEL
LIN {X 0,Y 512.411,Z 886.458,A -85,B 0,C 180,E1 22186.933,E2 22186.933} C_VEL
LIN {X 0,Y 514.793,Z 865.163,A -85,B 0,C 180,E1 22186.316,E2 22186.316} C_VEL
LIN {X 0,Y 516.918,Z 840.547,A -85,B 0,C 180,E1 22185.77,E2 22185.77} C_VEL
LIN {X 0,Y 519.086,Z 787.879,A -85,B 0,C 180,E1 22184.96,E2 22184.96} C_VEL
LIN {X 0,Y 527.339,Z 570.067,A -85,B 0,C 180,E1 22181.714,E2 22181.714} C_VEL
LIN {X 0,Y 528.751,Z 532.081,A -85,B 0,C 180,E1 22181.136,E2 22181.136} C_VEL
LIN {X 0,Y 516.831,Z 511.042,A -85,B 0,C 180,E1 22179.245,E2 22179.245} C_VEL
LIN {X 0,Y 505.116,Z 492.034,A -85,B 0,C 180,E1 22177.264,E2 22177.264} C_VEL
LIN {X 0,Y 493.184,Z 474.029,A -85,B 0,C 180,E1 22175.084,E2 22175.084} C_VEL
LIN {X 0,Y 482.355,Z 458.77,A -85,B 0,C 180,E1 22172.931,E2 22172.931} C_VEL
LIN {X 0,Y 474.196,Z 447.898,A -85,B 0,C 180,E1 22171.176,E2 22171.176} C_VEL
LIN {X 0,Y 469.517,Z 441.736,A -85,B 0,C 180,E1 22170.066,E2 22170.066} C_VEL
LIN {X 0,Y 467.824,Z 438.092,A -85,B 0,C 180,E1 22169.164,E2 22169.164} C_VEL
LIN {X 0,Y 466.181,Z 434.331,A -85,B 0,C 180,E1 22168.113,E2 22168.113} C_VEL
LIN {X 0,Y 466.165,Z 434.12,A -85,B 0,C 180,E1 22164.455,E2 22164.455} C_VEL
LIN {X 0,Y 466.166,Z 434.149,A -85,B 0,C 180,E1 22160.858,E2 22160.858} C_VEL
LIN {X 0,Y 466.169,Z 434.154,A -85,B 0,C 180,E1 22157.217,E2 22157.217} C_VEL
LIN {X 0,Y 466.168,Z 434.121,A -85,B 0,C 180,E1 22153.521,E2 22153.521} C_VEL
LIN {X 0,Y 466.167,Z 434.13,A -85,B 0,C 180,E1 22149.881,E2 22149.881} C_VEL
LIN {X 0,Y 466.174,Z 434.161,A -85,B 0,C 180,E1 22146.157,E2 22146.157} C_VEL
LIN {X 0,Y 466.149,Z 434.123,A -85,B 0,C 180,E1 22142.459,E2 22142.459} C_VEL
LIN {X 0,Y 466.147,Z 434.134,A -85,B 0,C 180,E1 22138.771,E2 22138.771} C_VEL
LIN {X 0,Y 466.159,Z 434.16,A -85,B 0,C 180,E1 22135.078,E2 22135.078} C_VEL
LIN {X 0,Y 466.173,Z 434.116,A -85,B 0,C 180,E1 22131.489,E2 22131.489} C_VEL
LIN {X 0,Y 466.155,Z 434.139,A -85,B 0,C 180,E1 22127.865,E2 22127.865} C_VEL
LIN {X 0,Y 466.131,Z 434.156,A -85,B 0,C 180,E1 22124.319,E2 22124.319} C_VEL
LIN {X 0,Y 466.132,Z 434.125,A -85,B 0,C 180,E1 22120.707,E2 22120.707} C_VEL
LIN {X 0,Y 466.171,Z 434.13,A -85,B 0,C 180,E1 22117.156,E2 22117.156} C_VEL
LIN {X 0,Y 466.159,Z 434.161,A -85,B 0,C 180,E1 22113.438,E2 22113.438} C_VEL
LIN {X 0,Y 466.113,Z 434.148,A -85,B 0,C 180,E1 22110.011,E2 22110.011} C_VEL
LIN {X 0,Y 466.18,Z 434.399,A -85,B 0,C 180,E1 22107.428,E2 22107.428} C_VEL
LIN {X 0,Y 466.621,Z 435.984,A -85,B 0,C 180,E1 22107.122,E2 22107.122} C_VEL
LIN {X 0,Y 468.47,Z 438.866,A -85,B 0,C 180,E1 22106.66,E2 22106.66} C_VEL
LIN {X 0,Y 470.989,Z 440.815,A -85,B 0,C 180,E1 22106.107,E2 22106.107} C_VEL
LIN {X 0,Y 473.323,Z 444.536,A -85,B 0,C 180,E1 22105.554,E2 22105.554} C_VEL
LIN {X 0,Y 475.912,Z 447.08,A -85,B 0,C 180,E1 22105,E2 22105} C_VEL
LIN {X 0,Y 478.945,Z 451.16,A -85,B 0,C 180,E1 22104.339,E2 22104.339} C_VEL
LIN {X 0,Y 480.708,Z 453.074,A -85,B 0,C 180,E1 22103.975,E2 22103.975} C_VEL
LIN {X 0,Y 484.363,Z 457.611,A -85,B 0,C 180,E1 22103.226,E2 22103.226} C_VEL
LIN {X 0,Y 496.977,Z 474.031,A -85,B 0,C 180,E1 22100.802,E2 22100.802} C_VEL
LIN {X 0,Y 508.335,Z 489.827,A -85,B 0,C 180,E1 22098.799,E2 22098.799} C_VEL
LIN {X 0,Y 520.431,Z 507.672,A -85,B 0,C 180,E1 22096.826,E2 22096.826} C_VEL
LIN {X 0,Y 529.075,Z 521.491,A -85,B 0,C 180,E1 22095.494,E2 22095.494} C_VEL
LIN {X 0,Y 519.585,Z 765.228,A -85,B 0,C 180,E1 22091.872,E2 22091.872} C_VEL
LIN {X 0,Y 517.533,Z 814.324,A -85,B 0,C 180,E1 22091.111,E2 22091.111} C_VEL
LIN {X 0,Y 515.591,Z 838.342,A -85,B 0,C 180,E1 22090.558,E2 22090.558} C_VEL
LIN {X 0,Y 513.2,Z 861.35,A -85,B 0,C 180,E1 22089.863,E2 22089.863} C_VEL
LIN {X 0,Y 510.223,Z 883.965,A -85,B 0,C 180,E1 22088.982,E2 22088.982} C_VEL
LIN {X 0,Y 507.157,Z 904.07,A -85,B 0,C 180,E1 22088.033,E2 22088.033} C_VEL
LIN {X 0,Y 502.994,Z 927.883,A -85,B 0,C 180,E1 22086.681,E2 22086.681} C_VEL
LIN {X 0,Y 499.345,Z 946.615,A -85,B 0,C 180,E1 22085.414,E2 22085.414} C_VEL
LIN {X 0,Y 495.059,Z 967.104,A -85,B 0,C 180,E1 22083.81,E2 22083.81} C_VEL
LIN {X 0,Y 490.862,Z 985.491,A -85,B 0,C 180,E1 22082.118,E2 22082.118} C_VEL
LIN {X 0,Y 486.662,Z 1003.468,A -85,B 0,C 180,E1 22080.224,E2 22080.224} C_VEL
LIN {X 0,Y 482.41,Z 1020.936,A -85,B 0,C 180,E1 22078.067,E2 22078.067} C_VEL
LIN {X 0,Y 478.877,Z 1035.531,A -85,B 0,C 180,E1 22076.007,E2 22076.007} C_VEL
LIN {X 0,Y 475.076,Z 1051.339,A -85,B 0,C 180,E1 22073.415,E2 22073.415} C_VEL
LIN {X 0,Y 474.375,Z 1054.367,A -85,B 0,C 180,E1 22072.87,E2 22072.87} C_VEL
LIN {X 0,Y 472.478,Z 1058.695,A -85,B 0,C 180,E1 22072.122,E2 22072.122} C_VEL
LIN {X 0,Y 464.443,Z 1069.275,A -85,B 0,C 180,E1 22070.269,E2 22070.269} C_VEL
LIN {X 0,Y 462.655,Z 1073.083,A -85,B 0,C 180,E1 22069.465,E2 22069.465} C_VEL
LIN {X 0,Y 460.238,Z 1084.547,A -85,B 0,C 180,E1 22066.535,E2 22066.535} C_VEL
LIN {X 0,Y 458.691,Z 1092.931,A -85,B 0,C 180,E1 22064.003,E2 22064.003} C_VEL
LIN {X 0,Y 457.35,Z 1101.583,A -85,B 0,C 180,E1 22060.837,E2 22060.837} C_VEL
LIN {X 0,Y 456.661,Z 1107.344,A -85,B 0,C 180,E1 22058.182,E2 22058.182} C_VEL
LIN {X 0,Y 456.222,Z 1112.482,A -85,B 0,C 180,E1 22055.156,E2 22055.156} C_VEL
LIN {X 0,Y 456.043,Z 1115.745,A -85,B 0,C 180,E1 22052.262,E2 22052.262} C_VEL
LIN {X 0,Y 455.99,Z 1117.569,A -85,B 0,C 180,E1 22049.623,E2 22049.623} C_VEL
LIN {X 0,Y 455.96,Z 1118.228,A -85,B 0,C 180,E1 22046.48,E2 22046.48} C_VEL
LIN {X 0,Y 456,Z 1117.44,A -85,B 0,C 180,E1 22043.832,E2 22043.832} C_VEL
LIN {X 0,Y 456.075,Z 1115.524,A -85,B 0,C 180,E1 22041.172,E2 22041.172} C_VEL
LIN {X 0,Y 456.316,Z 1111.644,A -85,B 0,C 180,E1 22037.985,E2 22037.985} C_VEL
LIN {X 0,Y 456.788,Z 1106.977,A -85,B 0,C 180,E1 22035.29,E2 22035.29} C_VEL
LIN {X 0,Y 457.72,Z 1100.301,A -85,B 0,C 180,E1 22032.26,E2 22032.26} C_VEL
LIN {X 0,Y 459.105,Z 1092.076,A -85,B 0,C 180,E1 22029.34,E2 22029.34} C_VEL
LIN {X 0,Y 461.059,Z 1082.513,A -85,B 0,C 180,E1 22026.482,E2 22026.482} C_VEL
LIN {X 0,Y 463.688,Z 1070.954,A -85,B 0,C 180,E1 22023.627,E2 22023.627} C_VEL
LIN {X 0,Y 466.749,Z 1058.817,A -85,B 0,C 180,E1 22021.043,E2 22021.043} C_VEL
LIN {X 0,Y 470.467,Z 1044.537,A -85,B 0,C 180,E1 22018.458,E2 22018.458} C_VEL
LIN {X 0,Y 474.125,Z 1030.926,A -85,B 0,C 180,E1 22016.313,E2 22016.313} C_VEL
LIN {X 0,Y 478.948,Z 1013.119,A -85,B 0,C 180,E1 22013.895,E2 22013.895} C_VEL
LIN {X 0,Y 483.103,Z 997.408,A -85,B 0,C 180,E1 22012.052,E2 22012.052} C_VEL
LIN {X 0,Y 487.998,Z 978.366,A -85,B 0,C 180,E1 22010.109,E2 22010.109} C_VEL
LIN {X 0,Y 492.507,Z 959.637,A -85,B 0,C 180,E1 22008.481,E2 22008.481} C_VEL
LIN {X 0,Y 497.187,Z 939.124,A -85,B 0,C 180,E1 22006.939,E2 22006.939} C_VEL
LIN {X 0,Y 501.324,Z 918.603,A -85,B 0,C 180,E1 22005.647,E2 22005.647} C_VEL
LIN {X 0,Y 504.904,Z 899.228,A -85,B 0,C 180,E1 22004.607,E2 22004.607} C_VEL
LIN {X 0,Y 508.799,Z 874.67,A -85,B 0,C 180,E1 22003.518,E2 22003.518} C_VEL
LIN {X 0,Y 511.528,Z 853.844,A -85,B 0,C 180,E1 22002.777,E2 22002.777} C_VEL
LIN {X 0,Y 514.155,Z 829.146,A -85,B 0,C 180,E1 22002.095,E2 22002.095} C_VEL
LIN {X 0,Y 515.778,Z 806.329,A -85,B 0,C 180,E1 22001.64,E2 22001.64} C_VEL
LIN {X 0,Y 526.332,Z 564.5,A -85,B 0,C 180,E1 21997.984,E2 21997.984} C_VEL
LIN {X 0,Y 527.938,Z 527.132,A -85,B 0,C 180,E1 21997.408,E2 21997.408} C_VEL
LIN {X 0,Y 516.313,Z 509.543,A -85,B 0,C 180,E1 21995.383,E2 21995.383} C_VEL
LIN {X 0,Y 504.067,Z 492.174,A -85,B 0,C 180,E1 21993.059,E2 21993.059} C_VEL
LIN {X 0,Y 494.815,Z 480.196,A -85,B 0,C 180,E1 21991.152,E2 21991.152} C_VEL
LIN {X 0,Y 487.178,Z 470.373,A -85,B 0,C 180,E1 21989.443,E2 21989.443} C_VEL
LIN {X 0,Y 483.049,Z 465.259,A -85,B 0,C 180,E1 21988.464,E2 21988.464} C_VEL
LIN {X 0,Y 479.372,Z 460.643,A -85,B 0,C 180,E1 21987.551,E2 21987.551} C_VEL
LIN {X 0,Y 475.126,Z 455.924,A -85,B 0,C 180,E1 21986.463,E2 21986.463} C_VEL
LIN {X 0,Y 473.822,Z 454.049,A -85,B 0,C 180,E1 21986.103,E2 21986.103} C_VEL
LIN {X 0,Y 470.538,Z 450.851,A -85,B 0,C 180,E1 21985.218,E2 21985.218} C_VEL
LIN {X 0,Y 468.647,Z 447.92,A -85,B 0,C 180,E1 21984.653,E2 21984.653} C_VEL
LIN {X 0,Y 465.399,Z 445.12,A -85,B 0,C 180,E1 21983.722,E2 21983.722} C_VEL
LIN {X 0,Y 463.375,Z 441.7,A -85,B 0,C 180,E1 21983.057,E2 21983.057} C_VEL
LIN {X 0,Y 459.996,Z 439.306,A -85,B 0,C 180,E1 21982.022,E2 21982.022} C_VEL
LIN {X 0,Y 458.325,Z 435.914,A -85,B 0,C 180,E1 21981.321,E2 21981.321} C_VEL
LIN {X 0,Y 458.23,Z 435.149,A -85,B 0,C 180,E1 21980.835,E2 21980.835} C_VEL
LIN {X 0,Y 458.196,Z 435.138,A -85,B 0,C 180,E1 21977.265,E2 21977.265} C_VEL
LIN {X 0,Y 458.193,Z 435.158,A -85,B 0,C 180,E1 21973.632,E2 21973.632} C_VEL
LIN {X 0,Y 458.208,Z 435.136,A -85,B 0,C 180,E1 21969.927,E2 21969.927} C_VEL
LIN {X 0,Y 458.235,Z 435.115,A -85,B 0,C 180,E1 21966.264,E2 21966.264} C_VEL
LIN {X 0,Y 458.226,Z 435.114,A -85,B 0,C 180,E1 21962.626,E2 21962.626} C_VEL
LIN {X 0,Y 458.216,Z 435.138,A -85,B 0,C 180,E1 21959,E2 21959} C_VEL
LIN {X 0,Y 458.214,Z 435.142,A -85,B 0,C 180,E1 21955.243,E2 21955.243} C_VEL
LIN {X 0,Y 458.218,Z 435.12,A -85,B 0,C 180,E1 21951.467,E2 21951.467} C_VEL
LIN {X 0,Y 458.229,Z 435.113,A -85,B 0,C 180,E1 21947.78,E2 21947.78} C_VEL
LIN {X 0,Y 458.226,Z 435.124,A -85,B 0,C 180,E1 21944.171,E2 21944.171} C_VEL
LIN {X 0,Y 458.23,Z 435.138,A -85,B 0,C 180,E1 21940.497,E2 21940.497} C_VEL
LIN {X 0,Y 458.259,Z 435.333,A -85,B 0,C 180,E1 21936.976,E2 21936.976} C_VEL
LIN {X 0,Y 459.864,Z 439.085,A -85,B 0,C 180,E1 21935.599,E2 21935.599} C_VEL
LIN {X 0,Y 461.538,Z 441.272,A -85,B 0,C 180,E1 21934.942,E2 21934.942} C_VEL
LIN {X 0,Y 464.807,Z 445.386,A -85,B 0,C 180,E1 21933.901,E2 21933.901} C_VEL
LIN {X 0,Y 466.789,Z 447.737,A -85,B 0,C 180,E1 21933.301,E2 21933.301} C_VEL
LIN {X 0,Y 474.993,Z 458.16,A -85,B 0,C 180,E1 21930.973,E2 21930.973} C_VEL
LIN {X 0,Y 479.492,Z 464.038,A -85,B 0,C 180,E1 21929.796,E2 21929.796} C_VEL
LIN {X 0,Y 486.602,Z 473.556,A -85,B 0,C 180,E1 21928.054,E2 21928.054} C_VEL
LIN {X 0,Y 494.644,Z 484.816,A -85,B 0,C 180,E1 21926.227,E2 21926.227} C_VEL
LIN {X 0,Y 503.803,Z 498.27,A -85,B 0,C 180,E1 21924.303,E2 21924.303} C_VEL
LIN {X 0,Y 515.039,Z 515.905,A -85,B 0,C 180,E1 21922.123,E2 21922.123} C_VEL
LIN {X 0,Y 526.653,Z 535.696,A -85,B 0,C 180,E1 21920.044,E2 21920.044} C_VEL
LIN {X 0,Y 527.784,Z 538.067,A -85,B 0,C 180,E1 21919.842,E2 21919.842} C_VEL
LIN {X 0,Y 518.3,Z 757.174,A -85,B 0,C 180,E1 21916.533,E2 21916.533} C_VEL
LIN {X 0,Y 514.776,Z 837.46,A -85,B 0,C 180,E1 21915.299,E2 21915.299} C_VEL
LIN {X 0,Y 512.508,Z 862.949,A -85,B 0,C 180,E1 21914.752,E2 21914.752} C_VEL
LIN {X 0,Y 510.058,Z 883.242,A -85,B 0,C 180,E1 21914.178,E2 21914.178} C_VEL
LIN {X 0,Y 506.563,Z 907.36,A -85,B 0,C 180,E1 21913.308,E2 21913.308} C_VEL
LIN {X 0,Y 502.993,Z 928.132,A -85,B 0,C 180,E1 21912.368,E2 21912.368} C_VEL
LIN {X 0,Y 499.011,Z 949.079,A -85,B 0,C 180,E1 21911.242,E2 21911.242} C_VEL
LIN {X 0,Y 494.287,Z 971.195,A -85,B 0,C 180,E1 21909.81,E2 21909.81} C_VEL
LIN {X 0,Y 490.109,Z 989.487,A -85,B 0,C 180,E1 21908.425,E2 21908.425} C_VEL
LIN {X 0,Y 484.837,Z 1011.123,A -85,B 0,C 180,E1 21906.511,E2 21906.511} C_VEL
LIN {X 0,Y 480.535,Z 1028.092,A -85,B 0,C 180,E1 21904.76,E2 21904.76} C_VEL
LIN {X 0,Y 475.775,Z 1046.69,A -85,B 0,C 180,E1 21902.548,E2 21902.548} C_VEL
LIN {X 0,Y 471.728,Z 1062.357,A -85,B 0,C 180,E1 21900.38,E2 21900.38} C_VEL
LIN {X 0,Y 467.827,Z 1077.992,A -85,B 0,C 180,E1 21897.909,E2 21897.909} C_VEL
LIN {X 0,Y 464.421,Z 1092.143,A -85,B 0,C 180,E1 21895.276,E2 21895.276} C_VEL
LIN {X 0,Y 461.646,Z 1104.937,A -85,B 0,C 180,E1 21892.543,E2 21892.543} C_VEL
LIN {X 0,Y 459.453,Z 1116.038,A -85,B 0,C 180,E1 21889.714,E2 21889.714} C_VEL
LIN {X 0,Y 457.966,Z 1125.173,A -85,B 0,C 180,E1 21887,E2 21887} C_VEL
LIN {X 0,Y 456.869,Z 1133.636,A -85,B 0,C 180,E1 21883.93,E2 21883.93} C_VEL
LIN {X 0,Y 456.328,Z 1139.354,A -85,B 0,C 180,E1 21881.374,E2 21881.374} C_VEL
LIN {X 0,Y 456.048,Z 1144.538,A -85,B 0,C 180,E1 21878.447,E2 21878.447} C_VEL
LIN {X 0,Y 455.944,Z 1148.012,A -85,B 0,C 180,E1 21875.537,E2 21875.537} C_VEL
LIN {X 0,Y 455.945,Z 1149.817,A -85,B 0,C 180,E1 21873.143,E2 21873.143} C_VEL
LIN {X 0,Y 455.952,Z 1150.647,A -85,B 0,C 180,E1 21870.628,E2 21870.628} C_VEL
LIN {X 0,Y 455.956,Z 1150.156,A -85,B 0,C 180,E1 21867.612,E2 21867.612} C_VEL
LIN {X 0,Y 455.942,Z 1148.343,A -85,B 0,C 180,E1 21864.967,E2 21864.967} C_VEL
LIN {X 0,Y 455.983,Z 1145.656,A -85,B 0,C 180,E1 21862.566,E2 21862.566} C_VEL
LIN {X 0,Y 456.195,Z 1141.074,A -85,B 0,C 180,E1 21859.646,E2 21859.646} C_VEL
LIN {X 0,Y 456.699,Z 1134.713,A -85,B 0,C 180,E1 21856.71,E2 21856.71} C_VEL
LIN {X 0,Y 457.519,Z 1127.549,A -85,B 0,C 180,E1 21854.016,E2 21854.016} C_VEL
LIN {X 0,Y 459.002,Z 1117.475,A -85,B 0,C 180,E1 21850.928,E2 21850.928} C_VEL
LIN {X 0,Y 460.761,Z 1107.492,A -85,B 0,C 180,E1 21848.351,E2 21848.351} C_VEL
LIN {X 0,Y 463.492,Z 1094.011,A -85,B 0,C 180,E1 21845.395,E2 21845.395} C_VEL
LIN {X 0,Y 466.198,Z 1081.781,A -85,B 0,C 180,E1 21843.093,E2 21843.093} C_VEL
LIN {X 0,Y 469.829,Z 1066.323,A -85,B 0,C 180,E1 21840.553,E2 21840.553} C_VEL
LIN {X 0,Y 473.558,Z 1050.716,A -85,B 0,C 180,E1 21838.352,E2 21838.352} C_VEL
LIN {X 0,Y 477.917,Z 1032.969,A -85,B 0,C 180,E1 21836.161,E2 21836.161} C_VEL
LIN {X 0,Y 482.263,Z 1014.532,A -85,B 0,C 180,E1 21834.219,E2 21834.219} C_VEL
LIN {X 0,Y 486.694,Z 995.475,A -85,B 0,C 180,E1 21832.469,E2 21832.469} C_VEL
LIN {X 0,Y 491.308,Z 974.228,A -85,B 0,C 180,E1 21830.816,E2 21830.816} C_VEL
LIN {X 0,Y 495.23,Z 954.933,A -85,B 0,C 180,E1 21829.524,E2 21829.524} C_VEL
LIN {X 0,Y 499.599,Z 931.356,A -85,B 0,C 180,E1 21828.205,E2 21828.205} C_VEL
LIN {X 0,Y 502.762,Z 911.935,A -85,B 0,C 180,E1 21827.298,E2 21827.298} C_VEL
LIN {X 0,Y 506.204,Z 888.088,A -85,B 0,C 180,E1 21826.385,E2 21826.385} C_VEL
LIN {X 0,Y 508.796,Z 865.728,A -85,B 0,C 180,E1 21825.727,E2 21825.727} C_VEL
LIN {X 0,Y 510.94,Z 842.046,A -85,B 0,C 180,E1 21825.19,E2 21825.19} C_VEL
LIN {X 0,Y 512.735,Z 802.682,A -85,B 0,C 180,E1 21824.564,E2 21824.564} C_VEL
LIN {X 0,Y 521.304,Z 584.245,A -85,B 0,C 180,E1 21821.286,E2 21821.286} C_VEL
LIN {X 0,Y 523.225,Z 535.391,A -85,B 0,C 180,E1 21820.541,E2 21820.541} C_VEL
LIN {X 0,Y 510.89,Z 513.738,A -85,B 0,C 180,E1 21818.526,E2 21818.526} C_VEL
LIN {X 0,Y 499.443,Z 495.113,A -85,B 0,C 180,E1 21816.52,E2 21816.52} C_VEL
LIN {X 0,Y 487.656,Z 477.463,A -85,B 0,C 180,E1 21814.288,E2 21814.288} C_VEL
LIN {X 0,Y 478.544,Z 464.563,A -85,B 0,C 180,E1 21812.415,E2 21812.415} C_VEL
LIN {X 0,Y 471.078,Z 454.5,A -85,B 0,C 180,E1 21810.766,E2 21810.766} C_VEL
LIN {X 0,Y 463.622,Z 444.759,A -85,B 0,C 180,E1 21808.994,E2 21808.994} C_VEL
LIN {X 0,Y 460.864,Z 440.923,A -85,B 0,C 180,E1 21808.228,E2 21808.228} C_VEL
LIN {X 0,Y 458.404,Z 436.061,A -85,B 0,C 180,E1 21806.841,E2 21806.841} C_VEL
LIN {X 0,Y 458.246,Z 435.248,A -85,B 0,C 180,E1 21806.54,E2 21806.54} C_VEL
LIN {X 0,Y 458.23,Z 435.118,A -85,B 0,C 180,E1 21802.856,E2 21802.856} C_VEL
LIN {X 0,Y 458.226,Z 435.11,A -85,B 0,C 180,E1 21799.106,E2 21799.106} C_VEL
LIN {X 0,Y 458.236,Z 435.123,A -85,B 0,C 180,E1 21795.439,E2 21795.439} C_VEL
LIN {X 0,Y 458.231,Z 435.15,A -85,B 0,C 180,E1 21791.709,E2 21791.709} C_VEL
LIN {X 0,Y 458.231,Z 435.109,A -85,B 0,C 180,E1 21787.901,E2 21787.901} C_VEL
LIN {X 0,Y 458.221,Z 435.116,A -85,B 0,C 180,E1 21784.255,E2 21784.255} C_VEL
LIN {X 0,Y 458.211,Z 435.154,A -85,B 0,C 180,E1 21780.625,E2 21780.625} C_VEL
LIN {X 0,Y 458.212,Z 435.107,A -85,B 0,C 180,E1 21776.998,E2 21776.998} C_VEL
LIN {X 0,Y 458.241,Z 435.121,A -85,B 0,C 180,E1 21773.359,E2 21773.359} C_VEL
LIN {X 0,Y 458.235,Z 435.147,A -85,B 0,C 180,E1 21769.565,E2 21769.565} C_VEL
LIN {X 0,Y 458.202,Z 435.109,A -85,B 0,C 180,E1 21765.982,E2 21765.982} C_VEL
LIN {X 0,Y 458.189,Z 435.127,A -85,B 0,C 180,E1 21762.342,E2 21762.342} C_VEL
LIN {X 0,Y 458.193,Z 435.156,A -85,B 0,C 180,E1 21758.627,E2 21758.627} C_VEL
LIN {X 0,Y 458.222,Z 435.117,A -85,B 0,C 180,E1 21755.093,E2 21755.093} C_VEL
LIN {X 0,Y 458.213,Z 435.114,A -85,B 0,C 180,E1 21751.452,E2 21751.452} C_VEL
LIN {X 0,Y 458.258,Z 435.307,A -85,B 0,C 180,E1 21749.152,E2 21749.152} C_VEL
LIN {X 0,Y 458.552,Z 436.683,A -85,B 0,C 180,E1 21748.828,E2 21748.828} C_VEL
LIN {X 0,Y 460.249,Z 439.592,A -85,B 0,C 180,E1 21748.355,E2 21748.355} C_VEL
LIN {X 0,Y 463.267,Z 441.929,A -85,B 0,C 180,E1 21747.638,E2 21747.638} C_VEL
LIN {X 0,Y 465.567,Z 445.648,A -85,B 0,C 180,E1 21747.05,E2 21747.05} C_VEL
LIN {X 0,Y 468.238,Z 448.147,A -85,B 0,C 180,E1 21746.44,E2 21746.44} C_VEL
LIN {X 0,Y 471.326,Z 452.319,A -85,B 0,C 180,E1 21745.719,E2 21745.719} C_VEL
LIN {X 0,Y 473.144,Z 454.307,A -85,B 0,C 180,E1 21745.319,E2 21745.319} C_VEL
LIN {X 0,Y 476.798,Z 458.787,A -85,B 0,C 180,E1 21744.523,E2 21744.523} C_VEL
LIN {X 0,Y 486.739,Z 471.628,A -85,B 0,C 180,E1 21742.476,E2 21742.476} C_VEL
LIN {X 0,Y 494.491,Z 481.892,A -85,B 0,C 180,E1 21740.996,E2 21740.996} C_VEL
LIN {X 0,Y 504.679,Z 496.145,A -85,B 0,C 180,E1 21739.17,E2 21739.17} C_VEL
LIN {X 0,Y 516.647,Z 513.988,A -85,B 0,C 180,E1 21737.176,E2 21737.176} C_VEL
LIN {X 0,Y 523.532,Z 525.25,A -85,B 0,C 180,E1 21736.084,E2 21736.084} C_VEL
LIN {X 0,Y 513.666,Z 769.671,A -85,B 0,C 180,E1 21732.426,E2 21732.426} C_VEL
LIN {X 0,Y 511.677,Z 815.015,A -85,B 0,C 180,E1 21731.713,E2 21731.713} C_VEL
LIN {X 0,Y 509.68,Z 838.855,A -85,B 0,C 180,E1 21731.158,E2 21731.158} C_VEL
LIN {X 0,Y 507.174,Z 862.22,A -85,B 0,C 180,E1 21730.445,E2 21730.445} C_VEL
LIN {X 0,Y 504.07,Z 884.892,A -85,B 0,C 180,E1 21729.55,E2 21729.55} C_VEL
LIN {X 0,Y 500.91,Z 904.923,A -85,B 0,C 180,E1 21728.594,E2 21728.594} C_VEL
LIN {X 0,Y 496.609,Z 928.623,A -85,B 0,C 180,E1 21727.232,E2 21727.232} C_VEL
LIN {X 0,Y 492.834,Z 947.35,A -85,B 0,C 180,E1 21725.951,E2 21725.951} C_VEL
LIN {X 0,Y 488.249,Z 968.387,A -85,B 0,C 180,E1 21724.276,E2 21724.276} C_VEL
LIN {X 0,Y 483.907,Z 986.748,A -85,B 0,C 180,E1 21722.559,E2 21722.559} C_VEL
LIN {X 0,Y 479.45,Z 1005.09,A -85,B 0,C 180,E1 21720.588,E2 21720.588} C_VEL
LIN {X 0,Y 475.285,Z 1021.468,A -85,B 0,C 180,E1 21718.526,E2 21718.526} C_VEL
LIN {X 0,Y 471.413,Z 1036.869,A -85,B 0,C 180,E1 21716.315,E2 21716.315} C_VEL
LIN {X 0,Y 467.572,Z 1052.112,A -85,B 0,C 180,E1 21713.756,E2 21713.756} C_VEL
LIN {X 0,Y 464.593,Z 1064.63,A -85,B 0,C 180,E1 21711.329,E2 21711.329} C_VEL
LIN {X 0,Y 462.655,Z 1073.083,A -85,B 0,C 180,E1 21709.465,E2 21709.465} C_VEL
LIN {X 0,Y 460.906,Z 1076.789,A -85,B 0,C 180,E1 21708.645,E2 21708.645} C_VEL
LIN {X 0,Y 452.948,Z 1086.094,A -85,B 0,C 180,E1 21706.465,E2 21706.465} C_VEL
LIN {X 0,Y 451.722,Z 1088.829,A -85,B 0,C 180,E1 21705.711,E2 21705.711} C_VEL
LIN {X 0,Y 450.097,Z 1097.697,A -85,B 0,C 180,E1 21702.705,E2 21702.705} C_VEL
LIN {X 0,Y 449.117,Z 1104.31,A -85,B 0,C 180,E1 21700,E2 21700} C_VEL
LIN {X 0,Y 448.433,Z 1110.432,A -85,B 0,C 180,E1 21696.787,E2 21696.787} C_VEL
LIN {X 0,Y 448.136,Z 1114.208,A -85,B 0,C 180,E1 21694.094,E2 21694.094} C_VEL
LIN {X 0,Y 447.999,Z 1117.059,A -85,B 0,C 180,E1 21691.151,E2 21691.151} C_VEL
LIN {X 0,Y 447.968,Z 1118.34,A -85,B 0,C 180,E1 21688.209,E2 21688.209} C_VEL
LIN {X 0,Y 447.969,Z 1118.376,A -85,B 0,C 180,E1 21685.648,E2 21685.648} C_VEL
LIN {X 0,Y 448,Z 1117.248,A -85,B 0,C 180,E1 21682.82,E2 21682.82} C_VEL
LIN {X 0,Y 448.166,Z 1114.401,A -85,B 0,C 180,E1 21679.707,E2 21679.707} C_VEL
LIN {X 0,Y 448.481,Z 1110.655,A -85,B 0,C 180,E1 21676.982,E2 21676.982} C_VEL
LIN {X 0,Y 449.231,Z 1104.552,A -85,B 0,C 180,E1 21673.713,E2 21673.713} C_VEL
LIN {X 0,Y 450.296,Z 1097.88,A -85,B 0,C 180,E1 21670.949,E2 21670.949} C_VEL
LIN {X 0,Y 452.05,Z 1089.035,A -85,B 0,C 180,E1 21667.912,E2 21667.912} C_VEL
LIN {X 0,Y 454.375,Z 1078.633,A -85,B 0,C 180,E1 21665.007,E2 21665.007} C_VEL
LIN {X 0,Y 457.319,Z 1067.112,A -85,B 0,C 180,E1 21662.244,E2 21662.244} C_VEL
LIN {X 0,Y 460.74,Z 1054.154,A -85,B 0,C 180,E1 21659.625,E2 21659.625} C_VEL
LIN {X 0,Y 464.45,Z 1040.893,A -85,B 0,C 180,E1 21657.291,E2 21657.291} C_VEL
LIN {X 0,Y 469.098,Z 1024.346,A -85,B 0,C 180,E1 21654.79,E2 21654.79} C_VEL
LIN {X 0,Y 473.425,Z 1008.907,A -85,B 0,C 180,E1 21652.773,E2 21652.773} C_VEL
LIN {X 0,Y 478.753,Z 989.451,A -85,B 0,C 180,E1 21650.586,E2 21650.586} C_VEL
LIN {X 0,Y 483.223,Z 972.286,A -85,B 0,C 180,E1 21648.93,E2 21648.93} C_VEL
LIN {X 0,Y 488.226,Z 952.049,A -85,B 0,C 180,E1 21647.241,E2 21647.241} C_VEL
LIN {X 0,Y 492.742,Z 931.73,A -85,B 0,C 180,E1 21645.809,E2 21645.809} C_VEL
LIN {X 0,Y 496.953,Z 911.304,A -85,B 0,C 180,E1 21644.58,E2 21644.58} C_VEL
LIN {X 0,Y 500.884,Z 889.144,A -85,B 0,C 180,E1 21643.478,E2 21643.478} C_VEL
LIN {X 0,Y 503.878,Z 869.732,A -85,B 0,C 180,E1 21642.674,E2 21642.674} C_VEL
LIN {X 0,Y 506.943,Z 846.072,A -85,B 0,C 180,E1 21641.882,E2 21641.882} C_VEL
LIN {X 0,Y 509.123,Z 823.528,A -85,B 0,C 180,E1 21641.315,E2 21641.315} C_VEL
LIN {X 0,Y 510.716,Z 799.809,A -85,B 0,C 180,E1 21640.872,E2 21640.872} C_VEL
LIN {X 0,Y 521.948,Z 550.007,A -85,B 0,C 180,E1 21637.083,E2 21637.083} C_VEL
LIN {X 0,Y 522.732,Z 530.913,A -85,B 0,C 180,E1 21636.778,E2 21636.778} C_VEL
LIN {X 0,Y 511.283,Z 513.66,A -85,B 0,C 180,E1 21634.721,E2 21634.721} C_VEL
LIN {X 0,Y 500.231,Z 497.989,A -85,B 0,C 180,E1 21632.561,E2 21632.561} C_VEL
LIN {X 0,Y 491.478,Z 486.46,A -85,B 0,C 180,E1 21630.707,E2 21630.707} C_VEL
LIN {X 0,Y 483.947,Z 476.742,A -85,B 0,C 180,E1 21628.98,E2 21628.98} C_VEL
LIN {X 0,Y 480.206,Z 472.069,A -85,B 0,C 180,E1 21628.072,E2 21628.072} C_VEL
LIN {X 0,Y 475.938,Z 466.801,A -85,B 0,C 180,E1 21626.987,E2 21626.987} C_VEL
LIN {X 0,Y 472.315,Z 462.485,A -85,B 0,C 180,E1 21626.024,E2 21626.024} C_VEL
LIN {X 0,Y 470.995,Z 460.968,A -85,B 0,C 180,E1 21625.663,E2 21625.663} C_VEL
LIN {X 0,Y 467.617,Z 457.151,A -85,B 0,C 180,E1 21624.711,E2 21624.711} C_VEL
LIN {X 0,Y 466.302,Z 455.232,A -85,B 0,C 180,E1 21624.312,E2 21624.312} C_VEL
LIN {X 0,Y 462.939,Z 452.001,A -85,B 0,C 180,E1 21623.316,E2 21623.316} C_VEL
LIN {X 0,Y 461.098,Z 449.101,A -85,B 0,C 180,E1 21622.706,E2 21622.706} C_VEL
LIN {X 0,Y 457.803,Z 446.447,A -85,B 0,C 180,E1 21621.661,E2 21621.661} C_VEL
LIN {X 0,Y 455.718,Z 442.798,A -85,B 0,C 180,E1 21620.888,E2 21620.888} C_VEL
LIN {X 0,Y 452.288,Z 440.533,A -85,B 0,C 180,E1 21619.703,E2 21619.703} C_VEL
LIN {X 0,Y 450.622,Z 437.66,A -85,B 0,C 180,E1 21619.004,E2 21619.004} C_VEL
LIN {X 0,Y 450.348,Z 436.491,A -85,B 0,C 180,E1 21618.646,E2 21618.646} C_VEL
LIN {X 0,Y 450.27,Z 436.119,A -85,B 0,C 180,E1 21617.045,E2 21617.045} C_VEL
LIN {X 0,Y 450.255,Z 436.142,A -85,B 0,C 180,E1 21613.424,E2 21613.424} C_VEL
LIN {X 0,Y 450.261,Z 436.13,A -85,B 0,C 180,E1 21609.717,E2 21609.717} C_VEL
LIN {X 0,Y 450.288,Z 436.105,A -85,B 0,C 180,E1 21606.119,E2 21606.119} C_VEL
LIN {X 0,Y 450.291,Z 436.099,A -85,B 0,C 180,E1 21602.418,E2 21602.418} C_VEL
LIN {X 0,Y 450.289,Z 436.115,A -85,B 0,C 180,E1 21598.728,E2 21598.728} C_VEL
LIN {X 0,Y 450.284,Z 436.137,A -85,B 0,C 180,E1 21594.904,E2 21594.904} C_VEL
LIN {X 0,Y 450.276,Z 436.114,A -85,B 0,C 180,E1 21591.181,E2 21591.181} C_VEL
LIN {X 0,Y 450.283,Z 436.103,A -85,B 0,C 180,E1 21587.431,E2 21587.431} C_VEL
LIN {X 0,Y 450.291,Z 436.106,A -85,B 0,C 180,E1 21583.752,E2 21583.752} C_VEL
LIN {X 0,Y 450.286,Z 436.108,A -85,B 0,C 180,E1 21580.003,E2 21580.003} C_VEL
LIN {X 0,Y 450.341,Z 436.457,A -85,B 0,C 180,E1 21579.123,E2 21579.123} C_VEL
LIN {X 0,Y 451.524,Z 439.477,A -85,B 0,C 180,E1 21578.091,E2 21578.091} C_VEL
LIN {X 0,Y 454.712,Z 443.004,A -85,B 0,C 180,E1 21576.889,E2 21576.889} C_VEL
LIN {X 0,Y 458.113,Z 446.897,A -85,B 0,C 180,E1 21575.705,E2 21575.705} C_VEL
LIN {X 0,Y 462.732,Z 452.759,A -85,B 0,C 180,E1 21574.189,E2 21574.189} C_VEL
LIN {X 0,Y 464.682,Z 455.184,A -85,B 0,C 180,E1 21573.584,E2 21573.584} C_VEL
LIN {X 0,Y 472.39,Z 465.05,A -85,B 0,C 180,E1 21571.352,E2 21571.352} C_VEL
LIN {X 0,Y 477.032,Z 471.249,A -85,B 0,C 180,E1 21570.11,E2 21570.11} C_VEL
LIN {X 0,Y 483.623,Z 480.132,A -85,B 0,C 180,E1 21568.461,E2 21568.461} C_VEL
LIN {X 0,Y 493.666,Z 494.386,A -85,B 0,C 180,E1 21566.152,E2 21566.152} C_VEL
LIN {X 0,Y 504.41,Z 510.778,A -85,B 0,C 180,E1 21563.897,E2 21563.897} C_VEL
LIN {X 0,Y 514.595,Z 527.457,A -85,B 0,C 180,E1 21561.926,E2 21561.926} C_VEL
LIN {X 0,Y 522.591,Z 541.53,A -85,B 0,C 180,E1 21560.472,E2 21560.472} C_VEL
LIN {X 0,Y 512.806,Z 759.824,A -85,B 0,C 180,E1 21557.153,E2 21557.153} C_VEL
LIN {X 0,Y 509.275,Z 837.279,A -85,B 0,C 180,E1 21555.954,E2 21555.954} C_VEL
LIN {X 0,Y 506.943,Z 862.703,A -85,B 0,C 180,E1 21555.406,E2 21555.406} C_VEL
LIN {X 0,Y 504.384,Z 883.255,A -85,B 0,C 180,E1 21554.822,E2 21554.822} C_VEL
LIN {X 0,Y 500.741,Z 907.521,A -85,B 0,C 180,E1 21553.94,E2 21553.94} C_VEL
LIN {X 0,Y 497.059,Z 928.238,A -85,B 0,C 180,E1 21552.995,E2 21552.995} C_VEL
LIN {X 0,Y 492.754,Z 950.143,A -85,B 0,C 180,E1 21551.805,E2 21551.805} C_VEL
LIN {X 0,Y 488.036,Z 971.299,A -85,B 0,C 180,E1 21550.414,E2 21550.414} C_VEL
LIN {X 0,Y 483.576,Z 990.133,A -85,B 0,C 180,E1 21548.971,E2 21548.971} C_VEL
LIN {X 0,Y 478.105,Z 1011.649,A -85,B 0,C 180,E1 21547.036,E2 21547.036} C_VEL
LIN {X 0,Y 473.647,Z 1028.545,A -85,B 0,C 180,E1 21545.266,E2 21545.266} C_VEL
LIN {X 0,Y 468.567,Z 1047.484,A -85,B 0,C 180,E1 21542.967,E2 21542.967} C_VEL
LIN {X 0,Y 464.471,Z 1062.706,A -85,B 0,C 180,E1 21540.821,E2 21540.821} C_VEL
LIN {X 0,Y 460.321,Z 1078.519,A -85,B 0,C 180,E1 21538.264,E2 21538.264} C_VEL
LIN {X 0,Y 457.045,Z 1091.516,A -85,B 0,C 180,E1 21535.808,E2 21535.808} C_VEL
LIN {X 0,Y 454.007,Z 1104.727,A -85,B 0,C 180,E1 21532.943,E2 21532.943} C_VEL
LIN {X 0,Y 451.686,Z 1115.815,A -85,B 0,C 180,E1 21530.067,E2 21530.067} C_VEL
LIN {X 0,Y 450.113,Z 1124.906,A -85,B 0,C 180,E1 21527.318,E2 21527.318} C_VEL
LIN {X 0,Y 448.933,Z 1133.389,A -85,B 0,C 180,E1 21524.182,E2 21524.182} C_VEL
LIN {X 0,Y 448.356,Z 1139.101,A -85,B 0,C 180,E1 21521.579,E2 21521.579} C_VEL
LIN {X 0,Y 448.055,Z 1144.276,A -85,B 0,C 180,E1 21518.599,E2 21518.599} C_VEL
LIN {X 0,Y 447.951,Z 1147.742,A -85,B 0,C 180,E1 21515.636,E2 21515.636} C_VEL
LIN {X 0,Y 447.951,Z 1149.541,A -85,B 0,C 180,E1 21513.199,E2 21513.199} C_VEL
LIN {X 0,Y 447.958,Z 1150.389,A -85,B 0,C 180,E1 21510.512,E2 21510.512} C_VEL
LIN {X 0,Y 447.953,Z 1149.792,A -85,B 0,C 180,E1 21507.441,E2 21507.441} C_VEL
LIN {X 0,Y 447.945,Z 1148.042,A -85,B 0,C 180,E1 21504.877,E2 21504.877} C_VEL
LIN {X 0,Y 447.984,Z 1145.347,A -85,B 0,C 180,E1 21502.433,E2 21502.433} C_VEL
LIN {X 0,Y 448.217,Z 1140.751,A -85,B 0,C 180,E1 21499.46,E2 21499.46} C_VEL
LIN {X 0,Y 448.757,Z 1134.378,A -85,B 0,C 180,E1 21496.47,E2 21496.47} C_VEL
LIN {X 0,Y 449.68,Z 1126.841,A -85,B 0,C 180,E1 21493.597,E2 21493.597} C_VEL
LIN {X 0,Y 451.202,Z 1117.111,A -85,B 0,C 180,E1 21490.585,E2 21490.585} C_VEL
LIN {X 0,Y 453.079,Z 1107.08,A -85,B 0,C 180,E1 21487.956,E2 21487.956} C_VEL
LIN {X 0,Y 456.012,Z 1093.324,A -85,B 0,C 180,E1 21484.902,E2 21484.902} C_VEL
LIN {X 0,Y 458.963,Z 1080.654,A -85,B 0,C 180,E1 21482.493,E2 21482.493} C_VEL
LIN {X 0,Y 463.117,Z 1063.73,A -85,B 0,C 180,E1 21479.726,E2 21479.726} C_VEL
LIN {X 0,Y 466.869,Z 1048.848,A -85,B 0,C 180,E1 21477.627,E2 21477.627} C_VEL
LIN {X 0,Y 471.659,Z 1029.845,A -85,B 0,C 180,E1 21475.305,E2 21475.305} C_VEL
LIN {X 0,Y 475.862,Z 1012.79,A -85,B 0,C 180,E1 21473.512,E2 21473.512} C_VEL
LIN {X 0,Y 480.668,Z 992.843,A -85,B 0,C 180,E1 21471.691,E2 21471.691} C_VEL
LIN {X 0,Y 485.155,Z 972.748,A -85,B 0,C 180,E1 21470.136,E2 21470.136} C_VEL
LIN {X 0,Y 489.648,Z 951.442,A -85,B 0,C 180,E1 21468.719,E2 21468.719} C_VEL
LIN {X 0,Y 493.75,Z 929.409,A -85,B 0,C 180,E1 21467.509,E2 21467.509} C_VEL
LIN {X 0,Y 497.02,Z 909.896,A -85,B 0,C 180,E1 21466.605,E2 21466.605} C_VEL
LIN {X 0,Y 500.621,Z 884.995,A -85,B 0,C 180,E1 21465.674,E2 21465.674} C_VEL
LIN {X 0,Y 503.086,Z 864.178,A -85,B 0,C 180,E1 21465.069,E2 21465.069} C_VEL
LIN {X 0,Y 505.308,Z 839.509,A -85,B 0,C 180,E1 21464.519,E2 21464.519} C_VEL
LIN {X 0,Y 507.73,Z 784.308,A -85,B 0,C 180,E1 21463.659,E2 21463.659} C_VEL
LIN {X 0,Y 516.669,Z 565.787,A -85,B 0,C 180,E1 21460.353,E2 21460.353} C_VEL
LIN {X 0,Y 517.677,Z 538.762,A -85,B 0,C 180,E1 21459.925,E2 21459.925} C_VEL
LIN {X 0,Y 506.394,Z 518.791,A -85,B 0,C 180,E1 21458.029,E2 21458.029} C_VEL
LIN {X 0,Y 495.031,Z 500.14,A -85,B 0,C 180,E1 21455.982,E2 21455.982} C_VEL
LIN {X 0,Y 482.733,Z 481.551,A -85,B 0,C 180,E1 21453.576,E2 21453.576} C_VEL
LIN {X 0,Y 471.853,Z 466.352,A -85,B 0,C 180,E1 21451.241,E2 21451.241} C_VEL
LIN {X 0,Y 467.749,Z 460.813,A -85,B 0,C 180,E1 21450.298,E2 21450.298} C_VEL
LIN {X 0,Y 460.969,Z 451.766,A -85,B 0,C 180,E1 21448.645,E2 21448.645} C_VEL
LIN {X 0,Y 456.396,Z 445.991,A -85,B 0,C 180,E1 21447.463,E2 21447.463} C_VEL
LIN {X 0,Y 453.156,Z 441.716,A -85,B 0,C 180,E1 21446.575,E2 21446.575} C_VEL
LIN {X 0,Y 451.143,Z 438.856,A -85,B 0,C 180,E1 21445.748,E2 21445.748} C_VEL
LIN {X 0,Y 450.317,Z 436.295,A -85,B 0,C 180,E1 21444.953,E2 21444.953} C_VEL
LIN {X 0,Y 450.299,Z 436.14,A -85,B 0,C 180,E1 21441.356,E2 21441.356} C_VEL
LIN {X 0,Y 450.291,Z 436.118,A -85,B 0,C 180,E1 21437.577,E2 21437.577} C_VEL
LIN {X 0,Y 450.286,Z 436.095,A -85,B 0,C 180,E1 21433.876,E2 21433.876} C_VEL
LIN {X 0,Y 450.29,Z 436.11,A -85,B 0,C 180,E1 21430.103,E2 21430.103} C_VEL
LIN {X 0,Y 450.287,Z 436.135,A -85,B 0,C 180,E1 21426.375,E2 21426.375} C_VEL
LIN {X 0,Y 450.268,Z 436.096,A -85,B 0,C 180,E1 21422.673,E2 21422.673} C_VEL
LIN {X 0,Y 450.278,Z 436.112,A -85,B 0,C 180,E1 21418.982,E2 21418.982} C_VEL
LIN {X 0,Y 450.291,Z 436.131,A -85,B 0,C 180,E1 21415.287,E2 21415.287} C_VEL
LIN {X 0,Y 450.296,Z 436.091,A -85,B 0,C 180,E1 21411.573,E2 21411.573} C_VEL
LIN {X 0,Y 450.272,Z 436.117,A -85,B 0,C 180,E1 21407.951,E2 21407.951} C_VEL
LIN {X 0,Y 450.254,Z 436.133,A -85,B 0,C 180,E1 21404.28,E2 21404.28} C_VEL
LIN {X 0,Y 450.248,Z 436.102,A -85,B 0,C 180,E1 21400.542,E2 21400.542} C_VEL
LIN {X 0,Y 450.275,Z 436.105,A -85,B 0,C 180,E1 21396.994,E2 21396.994} C_VEL
LIN {X 0,Y 450.291,Z 436.128,A -85,B 0,C 180,E1 21393.21,E2 21393.21} C_VEL
LIN {X 0,Y 450.309,Z 436.291,A -85,B 0,C 180,E1 21391.029,E2 21391.029} C_VEL
LIN {X 0,Y 450.644,Z 437.786,A -85,B 0,C 180,E1 21390.636,E2 21390.636} C_VEL
LIN {X 0,Y 452.404,Z 440.676,A -85,B 0,C 180,E1 21390.106,E2 21390.106} C_VEL
LIN {X 0,Y 455.434,Z 442.948,A -85,B 0,C 180,E1 21389.325,E2 21389.325} C_VEL
LIN {X 0,Y 457.662,Z 446.624,A -85,B 0,C 180,E1 21388.706,E2 21388.706} C_VEL
LIN {X 0,Y 460.664,Z 449.366,A -85,B 0,C 180,E1 21387.966,E2 21387.966} C_VEL
LIN {X 0,Y 463.609,Z 453.404,A -85,B 0,C 180,E1 21387.225,E2 21387.225} C_VEL
LIN {X 0,Y 465.595,Z 455.441,A -85,B 0,C 180,E1 21386.759,E2 21386.759} C_VEL
LIN {X 0,Y 469.095,Z 459.819,A -85,B 0,C 180,E1 21385.94,E2 21385.94} C_VEL
LIN {X 0,Y 475.472,Z 467.898,A -85,B 0,C 180,E1 21384.52,E2 21384.52} C_VEL
LIN {X 0,Y 483.235,Z 477.855,A -85,B 0,C 180,E1 21382.903,E2 21382.903} C_VEL
LIN {X 0,Y 493.824,Z 492.042,A -85,B 0,C 180,E1 21380.859,E2 21380.859} C_VEL
LIN {X 0,Y 507.061,Z 511.384,A -85,B 0,C 180,E1 21378.504,E2 21378.504} C_VEL
LIN {X 0,Y 518.061,Z 528.632,A -85,B 0,C 180,E1 21376.693,E2 21376.693} C_VEL
LIN {X 0,Y 507.85,Z 772.772,A -85,B 0,C 180,E1 21373.012,E2 21373.012} C_VEL
LIN {X 0,Y 505.879,Z 815.611,A -85,B 0,C 180,E1 21372.33,E2 21372.33} C_VEL
LIN {X 0,Y 503.821,Z 839.403,A -85,B 0,C 180,E1 21371.772,E2 21371.772} C_VEL
LIN {X 0,Y 501.256,Z 862.578,A -85,B 0,C 180,E1 21371.06,E2 21371.06} C_VEL
LIN {X 0,Y 497.967,Z 885.814,A -85,B 0,C 180,E1 21370.132,E2 21370.132} C_VEL
LIN {X 0,Y 494.529,Z 906.881,A -85,B 0,C 180,E1 21369.112,E2 21369.112} C_VEL
LIN {X 0,Y 490.272,Z 929.359,A -85,B 0,C 180,E1 21367.797,E2 21367.797} C_VEL
LIN {X 0,Y 486.368,Z 948.08,A -85,B 0,C 180,E1 21366.502,E2 21366.502} C_VEL
LIN {X 0,Y 481.495,Z 969.571,A -85,B 0,C 180,E1 21364.764,E2 21364.764} C_VEL
LIN {X 0,Y 477.161,Z 987.286,A -85,B 0,C 180,E1 21363.085,E2 21363.085} C_VEL
LIN {X 0,Y 472.52,Z 1005.639,A -85,B 0,C 180,E1 21361.086,E2 21361.086} C_VEL
LIN {X 0,Y 468.191,Z 1021.996,A -85,B 0,C 180,E1 21358.999,E2 21358.999} C_VEL
LIN {X 0,Y 463.964,Z 1038.204,A -85,B 0,C 180,E1 21356.632,E2 21356.632} C_VEL
LIN {X 0,Y 460.087,Z 1052.878,A -85,B 0,C 180,E1 21354.108,E2 21354.108} C_VEL
LIN {X 0,Y 456.762,Z 1066.327,A -85,B 0,C 180,E1 21351.443,E2 21351.443} C_VEL
LIN {X 0,Y 453.925,Z 1078.264,A -85,B 0,C 180,E1 21348.627,E2 21348.627} C_VEL
LIN {X 0,Y 451.853,Z 1088.085,A -85,B 0,C 180,E1 21345.926,E2 21345.926} C_VEL
LIN {X 0,Y 451.722,Z 1088.829,A -85,B 0,C 180,E1 21345.711,E2 21345.711} C_VEL
LIN {X 0,Y 450.219,Z 1091.915,A -85,B 0,C 180,E1 21344.826,E2 21344.826} C_VEL
LIN {X 0,Y 442.782,Z 1099.399,A -85,B 0,C 180,E1 21342.455,E2 21342.455} C_VEL
LIN {X 0,Y 441.7,Z 1101.396,A -85,B 0,C 180,E1 21341.641,E2 21341.641} C_VEL
LIN {X 0,Y 440.815,Z 1107.56,A -85,B 0,C 180,E1 21338.741,E2 21338.741} C_VEL
LIN {X 0,Y 440.315,Z 1112.38,A -85,B 0,C 180,E1 21335.865,E2 21335.865} C_VEL
LIN {X 0,Y 440.072,Z 1116.155,A -85,B 0,C 180,E1 21332.605,E2 21332.605} C_VEL
LIN {X 0,Y 440.006,Z 1118.041,A -85,B 0,C 180,E1 21329.87,E2 21329.87} C_VEL
LIN {X 0,Y 439.974,Z 1118.851,A -85,B 0,C 180,E1 21326.743,E2 21326.743} C_VEL
LIN {X 0,Y 440.014,Z 1118.04,A -85,B 0,C 180,E1 21323.738,E2 21323.738} C_VEL
LIN {X 0,Y 440.1,Z 1116.146,A -85,B 0,C 180,E1 21320.981,E2 21320.981} C_VEL
LIN {X 0,Y 440.386,Z 1112.311,A -85,B 0,C 180,E1 21317.677,E2 21317.677} C_VEL
LIN {X 0,Y 440.93,Z 1107.668,A -85,B 0,C 180,E1 21314.883,E2 21314.883} C_VEL
LIN {X 0,Y 441.97,Z 1101.187,A -85,B 0,C 180,E1 21311.808,E2 21311.808} C_VEL
LIN {X 0,Y 443.568,Z 1092.842,A -85,B 0,C 180,E1 21308.72,E2 21308.72} C_VEL
LIN {X 0,Y 445.755,Z 1083.307,A -85,B 0,C 180,E1 21305.764,E2 21305.764} C_VEL
LIN {X 0,Y 448.667,Z 1071.803,A -85,B 0,C 180,E1 21302.815,E2 21302.815} C_VEL
LIN {X 0,Y 452.044,Z 1059.698,A -85,B 0,C 180,E1 21300.153,E2 21300.153} C_VEL
LIN {X 0,Y 456.096,Z 1045.59,A -85,B 0,C 180,E1 21297.513,E2 21297.513} C_VEL
LIN {X 0,Y 460.119,Z 1031.911,A -85,B 0,C 180,E1 21295.294,E2 21295.294} C_VEL
LIN {X 0,Y 465.467,Z 1013.719,A -85,B 0,C 180,E1 21292.758,E2 21292.758} C_VEL
LIN {X 0,Y 470.102,Z 997.541,A -85,B 0,C 180,E1 21290.823,E2 21290.823} C_VEL
LIN {X 0,Y 475.674,Z 977.372,A -85,B 0,C 180,E1 21288.75,E2 21288.75} C_VEL
LIN {X 0,Y 480.308,Z 959.464,A -85,B 0,C 180,E1 21287.18,E2 21287.18} C_VEL
LIN {X 0,Y 485.402,Z 938.443,A -85,B 0,C 180,E1 21285.592,E2 21285.592} C_VEL
LIN {X 0,Y 489.785,Z 918.06,A -85,B 0,C 180,E1 21284.304,E2 21284.304} C_VEL
LIN {X 0,Y 493.901,Z 897.067,A -85,B 0,C 180,E1 21283.179,E2 21283.179} C_VEL
LIN {X 0,Y 497.729,Z 873.756,A -85,B 0,C 180,E1 21282.159,E2 21282.159} C_VEL
LIN {X 0,Y 500.528,Z 853.551,A -85,B 0,C 180,E1 21281.442,E2 21281.442} C_VEL
LIN {X 0,Y 503.356,Z 827.771,A -85,B 0,C 180,E1 21280.737,E2 21280.737} C_VEL
LIN {X 0,Y 504.974,Z 805.961,A -85,B 0,C 180,E1 21280.305,E2 21280.305} C_VEL
LIN {X 0,Y 516.48,Z 560.313,A -85,B 0,C 180,E1 21276.545,E2 21276.545} C_VEL
LIN {X 0,Y 517.586,Z 534.832,A -85,B 0,C 180,E1 21276.137,E2 21276.137} C_VEL
LIN {X 0,Y 505.947,Z 517.189,A -85,B 0,C 180,E1 21273.972,E2 21273.972} C_VEL
LIN {X 0,Y 496.075,Z 503.277,A -85,B 0,C 180,E1 21271.979,E2 21271.979} C_VEL
LIN {X 0,Y 486.238,Z 490.045,A -85,B 0,C 180,E1 21269.811,E2 21269.811} C_VEL
LIN {X 0,Y 477.607,Z 479.087,A -85,B 0,C 180,E1 21267.729,E2 21267.729} C_VEL
LIN {X 0,Y 473.07,Z 473.557,A -85,B 0,C 180,E1 21266.553,E2 21266.553} C_VEL
LIN {X 0,Y 468.615,Z 468.157,A -85,B 0,C 180,E1 21265.329,E2 21265.329} C_VEL
LIN {X 0,Y 465.102,Z 464.016,A -85,B 0,C 180,E1 21264.311,E2 21264.311} C_VEL
LIN {X 0,Y 463.782,Z 462.354,A -85,B 0,C 180,E1 21263.911,E2 21263.911} C_VEL
LIN {X 0,Y 460.416,Z 458.746,A -85,B 0,C 180,E1 21262.876,E2 21262.876} C_VEL
LIN {X 0,Y 459.032,Z 456.579,A -85,B 0,C 180,E1 21262.408,E2 21262.408} C_VEL
LIN {X 0,Y 455.712,Z 453.693,A -85,B 0,C 180,E1 21261.326,E2 21261.326} C_VEL
LIN {X 0,Y 453.548,Z 450.241,A -85,B 0,C 180,E1 21260.52,E2 21260.52} C_VEL
LIN {X 0,Y 450.366,Z 447.893,A -85,B 0,C 180,E1 21259.385,E2 21259.385} C_VEL
LIN {X 0,Y 448.408,Z 444.546,A -85,B 0,C 180,E1 21258.561,E2 21258.561} C_VEL
LIN {X 0,Y 447.578,Z 443.693,A -85,B 0,C 180,E1 21258.226,E2 21258.226} C_VEL
LIN {X 0,Y 444.421,Z 441.567,A -85,B 0,C 180,E1 21256.939,E2 21256.939} C_VEL
LIN {X 0,Y 442.57,Z 438.319,A -85,B 0,C 180,E1 21256,E2 21256} C_VEL
LIN {X 0,Y 442.323,Z 437.16,A -85,B 0,C 180,E1 21255.303,E2 21255.303} C_VEL
LIN {X 0,Y 442.316,Z 437.095,A -85,B 0,C 180,E1 21251.607,E2 21251.607} C_VEL
LIN {X 0,Y 442.332,Z 437.103,A -85,B 0,C 180,E1 21247.926,E2 21247.926} C_VEL
LIN {X 0,Y 442.356,Z 437.129,A -85,B 0,C 180,E1 21244.278,E2 21244.278} C_VEL
LIN {X 0,Y 442.359,Z 437.101,A -85,B 0,C 180,E1 21240.518,E2 21240.518} C_VEL
LIN {X 0,Y 442.342,Z 437.086,A -85,B 0,C 180,E1 21236.76,E2 21236.76} C_VEL
LIN {X 0,Y 442.336,Z 437.091,A -85,B 0,C 180,E1 21233.119,E2 21233.119} C_VEL
LIN {X 0,Y 442.341,Z 437.11,A -85,B 0,C 180,E1 21229.318,E2 21229.318} C_VEL
LIN {X 0,Y 442.354,Z 437.132,A -85,B 0,C 180,E1 21225.469,E2 21225.469} C_VEL
LIN {X 0,Y 442.377,Z 437.302,A -85,B 0,C 180,E1 21221.961,E2 21221.961} C_VEL
LIN {X 0,Y 442.658,Z 438.518,A -85,B 0,C 180,E1 21221.428,E2 21221.428} C_VEL
LIN {X 0,Y 444.37,Z 441.505,A -85,B 0,C 180,E1 21220.548,E2 21220.548} C_VEL
LIN {X 0,Y 447.646,Z 444.146,A -85,B 0,C 180,E1 21219.197,E2 21219.197} C_VEL
LIN {X 0,Y 451.63,Z 449.065,A -85,B 0,C 180,E1 21217.617,E2 21217.617} C_VEL
LIN {X 0,Y 457.219,Z 455.746,A -85,B 0,C 180,E1 21215.621,E2 21215.621} C_VEL
LIN {X 0,Y 460.856,Z 460.311,A -85,B 0,C 180,E1 21214.421,E2 21214.421} C_VEL
LIN {X 0,Y 469.711,Z 471.787,A -85,B 0,C 180,E1 21211.763,E2 21211.763} C_VEL
LIN {X 0,Y 474.898,Z 478.888,A -85,B 0,C 180,E1 21210.344,E2 21210.344} C_VEL
LIN {X 0,Y 480.776,Z 486.872,A -85,B 0,C 180,E1 21208.846,E2 21208.846} C_VEL
LIN {X 0,Y 491.624,Z 502.49,A -85,B 0,C 180,E1 21206.307,E2 21206.307} C_VEL
LIN {X 0,Y 503.032,Z 520.315,A -85,B 0,C 180,E1 21203.888,E2 21203.888} C_VEL
LIN {X 0,Y 514.215,Z 539.197,A -85,B 0,C 180,E1 21201.715,E2 21201.715} C_VEL
LIN {X 0,Y 517.451,Z 545.346,A -85,B 0,C 180,E1 21201.109,E2 21201.109} C_VEL
LIN {X 0,Y 507.286,Z 764.507,A -85,B 0,C 180,E1 21197.756,E2 21197.756} C_VEL
LIN {X 0,Y 503.842,Z 837.128,A -85,B 0,C 180,E1 21196.623,E2 21196.623} C_VEL
LIN {X 0,Y 501.453,Z 862.401,A -85,B 0,C 180,E1 21196.076,E2 21196.076} C_VEL
LIN {X 0,Y 498.782,Z 883.233,A -85,B 0,C 180,E1 21195.481,E2 21195.481} C_VEL
LIN {X 0,Y 494.982,Z 907.687,A -85,B 0,C 180,E1 21194.586,E2 21194.586} C_VEL
LIN {X 0,Y 491.187,Z 928.348,A -85,B 0,C 180,E1 21193.638,E2 21193.638} C_VEL
LIN {X 0,Y 486.746,Z 950.204,A -85,B 0,C 180,E1 21192.44,E2 21192.44} C_VEL
LIN {X 0,Y 481.895,Z 971.18,A -85,B 0,C 180,E1 21191.05,E2 21191.05} C_VEL
LIN {X 0,Y 477.373,Z 989.61,A -85,B 0,C 180,E1 21189.628,E2 21189.628} C_VEL
LIN {X 0,Y 471.755,Z 1010.958,A -85,B 0,C 180,E1 21187.697,E2 21187.697} C_VEL
LIN {X 0,Y 467.105,Z 1027.886,A -85,B 0,C 180,E1 21185.911,E2 21185.911} C_VEL
LIN {X 0,Y 461.922,Z 1046.416,A -85,B 0,C 180,E1 21183.652,E2 21183.652} C_VEL
LIN {X 0,Y 457.612,Z 1061.703,A -85,B 0,C 180,E1 21181.481,E2 21181.481} C_VEL
LIN {X 0,Y 453.442,Z 1076.908,A -85,B 0,C 180,E1 21179.021,E2 21179.021} C_VEL
LIN {X 0,Y 449.702,Z 1090.899,A -85,B 0,C 180,E1 21176.356,E2 21176.356} C_VEL
LIN {X 0,Y 446.643,Z 1103.378,A -85,B 0,C 180,E1 21173.624,E2 21173.624} C_VEL
LIN {X 0,Y 444.135,Z 1114.661,A -85,B 0,C 180,E1 21170.699,E2 21170.699} C_VEL
LIN {X 0,Y 442.474,Z 1123.439,A -85,B 0,C 180,E1 21168.035,E2 21168.035} C_VEL
LIN {X 0,Y 441.086,Z 1132.524,A -85,B 0,C 180,E1 21164.708,E2 21164.708} C_VEL
LIN {X 0,Y 440.413,Z 1138.589,A -85,B 0,C 180,E1 21161.923,E2 21161.923} C_VEL
LIN {X 0,Y 440.062,Z 1143.818,A -85,B 0,C 180,E1 21158.888,E2 21158.888} C_VEL
LIN {X 0,Y 439.965,Z 1147.355,A -85,B 0,C 180,E1 21155.87,E2 21155.87} C_VEL
LIN {X 0,Y 439.956,Z 1149.266,A -85,B 0,C 180,E1 21153.257,E2 21153.257} C_VEL
LIN {X 0,Y 439.963,Z 1150.108,A -85,B 0,C 180,E1 21150.521,E2 21150.521} C_VEL
LIN {X 0,Y 439.961,Z 1149.567,A -85,B 0,C 180,E1 21147.525,E2 21147.525} C_VEL
LIN {X 0,Y 439.948,Z 1147.856,A -85,B 0,C 180,E1 21144.915,E2 21144.915} C_VEL
LIN {X 0,Y 439.986,Z 1145.201,A -85,B 0,C 180,E1 21142.426,E2 21142.426} C_VEL
LIN {X 0,Y 440.207,Z 1140.875,A -85,B 0,C 180,E1 21139.53,E2 21139.53} C_VEL
LIN {X 0,Y 440.75,Z 1134.665,A -85,B 0,C 180,E1 21136.487,E2 21136.487} C_VEL
LIN {X 0,Y 441.637,Z 1127.583,A -85,B 0,C 180,E1 21133.695,E2 21133.695} C_VEL
LIN {X 0,Y 443.329,Z 1117.214,A -85,B 0,C 180,E1 21130.363,E2 21130.363} C_VEL
LIN {X 0,Y 445.291,Z 1107.234,A -85,B 0,C 180,E1 21127.689,E2 21127.689} C_VEL
LIN {X 0,Y 448.28,Z 1093.863,A -85,B 0,C 180,E1 21124.643,E2 21124.643} C_VEL
LIN {X 0,Y 451.411,Z 1080.958,A -85,B 0,C 180,E1 21122.136,E2 21122.136} C_VEL
LIN {X 0,Y 455.4,Z 1065.448,A -85,B 0,C 180,E1 21119.523,E2 21119.523} C_VEL
LIN {X 0,Y 459.486,Z 1049.81,A -85,B 0,C 180,E1 21117.264,E2 21117.264} C_VEL
LIN {X 0,Y 464.158,Z 1032.185,A -85,B 0,C 180,E1 21115.039,E2 21115.039} C_VEL
LIN {X 0,Y 468.914,Z 1013.522,A -85,B 0,C 180,E1 21113.035,E2 21113.035} C_VEL
LIN {X 0,Y 473.877,Z 993.767,A -85,B 0,C 180,E1 21111.194,E2 21111.194} C_VEL
LIN {X 0,Y 478.683,Z 972.994,A -85,B 0,C 180,E1 21109.565,E2 21109.565} C_VEL
LIN {X 0,Y 483.079,Z 952.808,A -85,B 0,C 180,E1 21108.203,E2 21108.203} C_VEL
LIN {X 0,Y 487.525,Z 929.978,A -85,B 0,C 180,E1 21106.924,E2 21106.924} C_VEL
LIN {X 0,Y 490.912,Z 910.452,A -85,B 0,C 180,E1 21106.008,E2 21106.008} C_VEL
LIN {X 0,Y 494.619,Z 885.846,A -85,B 0,C 180,E1 21105.072,E2 21105.072} C_VEL
LIN {X 0,Y 497.238,Z 864.437,A -85,B 0,C 180,E1 21104.443,E2 21104.443} C_VEL
LIN {X 0,Y 499.534,Z 840.045,A -85,B 0,C 180,E1 21103.891,E2 21103.891} C_VEL
LIN {X 0,Y 501.866,Z 789.309,A -85,B 0,C 180,E1 21103.09,E2 21103.09} C_VEL
LIN {X 0,Y 511.109,Z 571.186,A -85,B 0,C 180,E1 21099.766,E2 21099.766} C_VEL
LIN {X 0,Y 512.308,Z 542.277,A -85,B 0,C 180,E1 21099.315,E2 21099.315} C_VEL
LIN {X 0,Y 500.525,Z 521.365,A -85,B 0,C 180,E1 21097.268,E2 21097.268} C_VEL
LIN {X 0,Y 489.487,Z 503.421,A -85,B 0,C 180,E1 21095.209,E2 21095.209} C_VEL
LIN {X 0,Y 478.978,Z 487.443,A -85,B 0,C 180,E1 21093.086,E2 21093.086} C_VEL
LIN {X 0,Y 468.853,Z 473.065,A -85,B 0,C 180,E1 21090.857,E2 21090.857} C_VEL
LIN {X 0,Y 461.2,Z 462.582,A -85,B 0,C 180,E1 21089.019,E2 21089.019} C_VEL
LIN {X 0,Y 453.925,Z 453.129,A -85,B 0,C 180,E1 21087.128,E2 21087.128} C_VEL
LIN {X 0,Y 450.415,Z 448.433,A -85,B 0,C 180,E1 21086.146,E2 21086.146} C_VEL
LIN {X 0,Y 446.183,Z 443.379,A -85,B 0,C 180,E1 21084.917,E2 21084.917} C_VEL
LIN {X 0,Y 442.992,Z 439.391,A -85,B 0,C 180,E1 21083.83,E2 21083.83} C_VEL
LIN {X 0,Y 442.38,Z 437.289,A -85,B 0,C 180,E1 21083.159,E2 21083.159} C_VEL
LIN {X 0,Y 442.35,Z 437.086,A -85,B 0,C 180,E1 21079.407,E2 21079.407} C_VEL
LIN {X 0,Y 442.353,Z 437.103,A -85,B 0,C 180,E1 21075.604,E2 21075.604} C_VEL
LIN {X 0,Y 442.354,Z 437.122,A -85,B 0,C 180,E1 21071.832,E2 21071.832} C_VEL
LIN {X 0,Y 442.354,Z 437.082,A -85,B 0,C 180,E1 21068.056,E2 21068.056} C_VEL
LIN {X 0,Y 442.338,Z 437.094,A -85,B 0,C 180,E1 21064.408,E2 21064.408} C_VEL
LIN {X 0,Y 442.333,Z 437.129,A -85,B 0,C 180,E1 21060.648,E2 21060.648} C_VEL
LIN {X 0,Y 442.33,Z 437.084,A -85,B 0,C 180,E1 21056.89,E2 21056.89} C_VEL
LIN {X 0,Y 442.355,Z 437.094,A -85,B 0,C 180,E1 21053.25,E2 21053.25} C_VEL
LIN {X 0,Y 442.357,Z 437.126,A -85,B 0,C 180,E1 21049.45,E2 21049.45} C_VEL
LIN {X 0,Y 442.342,Z 437.084,A -85,B 0,C 180,E1 21045.736,E2 21045.736} C_VEL
LIN {X 0,Y 442.315,Z 437.097,A -85,B 0,C 180,E1 21042.095,E2 21042.095} C_VEL
LIN {X 0,Y 442.308,Z 437.135,A -85,B 0,C 180,E1 21038.378,E2 21038.378} C_VEL
LIN {X 0,Y 442.314,Z 437.104,A -85,B 0,C 180,E1 21034.707,E2 21034.707} C_VEL
LIN {X 0,Y 442.378,Z 437.393,A -85,B 0,C 180,E1 21032.979,E2 21032.979} C_VEL
LIN {X 0,Y 442.796,Z 439.025,A -85,B 0,C 180,E1 21032.607,E2 21032.607} C_VEL
LIN {X 0,Y 444.554,Z 441.738,A -85,B 0,C 180,E1 21032.033,E2 21032.033} C_VEL
LIN {X 0,Y 447.659,Z 444.016,A -85,B 0,C 180,E1 21031.154,E2 21031.154} C_VEL
LIN {X 0,Y 449.797,Z 447.601,A -85,B 0,C 180,E1 21030.502,E2 21030.502} C_VEL
LIN {X 0,Y 452.955,Z 450.429,A -85,B 0,C 180,E1 21029.656,E2 21029.656} C_VEL
LIN {X 0,Y 455.747,Z 454.36,A -85,B 0,C 180,E1 21028.89,E2 21028.89} C_VEL
LIN {X 0,Y 458.095,Z 456.631,A -85,B 0,C 180,E1 21028.299,E2 21028.299} C_VEL
LIN {X 0,Y 461.497,Z 460.961,A -85,B 0,C 180,E1 21027.439,E2 21027.439} C_VEL
LIN {X 0,Y 463.253,Z 463.084,A -85,B 0,C 180,E1 21027.012,E2 21027.012} C_VEL
LIN {X 0,Y 467.904,Z 468.901,A -85,B 0,C 180,E1 21025.915,E2 21025.915} C_VEL
LIN {X 0,Y 472.938,Z 475.303,A -85,B 0,C 180,E1 21024.784,E2 21024.784} C_VEL
LIN {X 0,Y 480.258,Z 484.799,A -85,B 0,C 180,E1 21023.232,E2 21023.232} C_VEL
LIN {X 0,Y 490.482,Z 498.651,A -85,B 0,C 180,E1 21021.218,E2 21021.218} C_VEL
LIN {X 0,Y 504.783,Z 519.733,A -85,B 0,C 180,E1 21018.635,E2 21018.635} C_VEL
LIN {X 0,Y 512.634,Z 532.413,A -85,B 0,C 180,E1 21017.309,E2 21017.309} C_VEL
LIN {X 0,Y 501.993,Z 778.156,A -85,B 0,C 180,E1 21013.578,E2 21013.578} C_VEL
LIN {X 0,Y 500.111,Z 816.567,A -85,B 0,C 180,E1 21012.953,E2 21012.953} C_VEL
LIN {X 0,Y 498.029,Z 839.863,A -85,B 0,C 180,E1 21012.402,E2 21012.402} C_VEL
LIN {X 0,Y 495.292,Z 863.82,A -85,B 0,C 180,E1 21011.657,E2 21011.657} C_VEL
LIN {X 0,Y 491.917,Z 886.731,A -85,B 0,C 180,E1 21010.729,E2 21010.729} C_VEL
LIN {X 0,Y 488.147,Z 909.091,A -85,B 0,C 180,E1 21009.63,E2 21009.63} C_VEL
LIN {X 0,Y 483.799,Z 930.977,A -85,B 0,C 180,E1 21008.318,E2 21008.318} C_VEL
LIN {X 0,Y 479.662,Z 950.122,A -85,B 0,C 180,E1 21006.97,E2 21006.97} C_VEL
LIN {X 0,Y 474.561,Z 971.602,A -85,B 0,C 180,E1 21005.188,E2 21005.188} C_VEL
LIN {X 0,Y 470.22,Z 988.732,A -85,B 0,C 180,E1 21003.533,E2 21003.533} C_VEL
LIN {X 0,Y 464.924,Z 1008.667,A -85,B 0,C 180,E1 21001.291,E2 21001.291} C_VEL
LIN {X 0,Y 460.659,Z 1024.29,A -85,B 0,C 180,E1 20999.241,E2 20999.241} C_VEL
LIN {X 0,Y 456.08,Z 1040.974,A -85,B 0,C 180,E1 20996.707,E2 20996.707} C_VEL
LIN {X 0,Y 452.524,Z 1053.998,A -85,B 0,C 180,E1 20994.406,E2 20994.406} C_VEL
LIN {X 0,Y 449.074,Z 1067.36,A -85,B 0,C 180,E1 20991.692,E2 20991.692} C_VEL
LIN {X 0,Y 446.247,Z 1078.69,A -85,B 0,C 180,E1 20988.959,E2 20988.959} C_VEL
LIN {X 0,Y 443.99,Z 1088.943,A -85,B 0,C 180,E1 20986.081,E2 20986.081} C_VEL
LIN {X 0,Y 442.28,Z 1097.736,A -85,B 0,C 180,E1 20983.066,E2 20983.066} C_VEL
LIN {X 0,Y 441.7,Z 1101.396,A -85,B 0,C 180,E1 20981.641,E2 20981.641} C_VEL
LIN {X 0,Y 440.368,Z 1103.638,A -85,B 0,C 180,E1 20980.69,E2 20980.69} C_VEL
LIN {X 0,Y 433.314,Z 1109.415,A -85,B 0,C 180,E1 20978.087,E2 20978.087} C_VEL
LIN {X 0,Y 432.536,Z 1110.717,A -85,B 0,C 180,E1 20977.302,E2 20977.302} C_VEL
LIN {X 0,Y 432.195,Z 1114.552,A -85,B 0,C 180,E1 20974.512,E2 20974.512} C_VEL
LIN {X 0,Y 432.033,Z 1117.356,A -85,B 0,C 180,E1 20971.591,E2 20971.591} C_VEL
LIN {X 0,Y 431.971,Z 1118.877,A -85,B 0,C 180,E1 20968.408,E2 20968.408} C_VEL
LIN {X 0,Y 431.98,Z 1118.977,A -85,B 0,C 180,E1 20965.752,E2 20965.752} C_VEL
LIN {X 0,Y 432.011,Z 1118.046,A -85,B 0,C 180,E1 20963.087,E2 20963.087} C_VEL
LIN {X 0,Y 432.171,Z 1115.529,A -85,B 0,C 180,E1 20959.873,E2 20959.873} C_VEL
LIN {X 0,Y 432.528,Z 1111.735,A -85,B 0,C 180,E1 20956.906,E2 20956.906} C_VEL
LIN {X 0,Y 433.229,Z 1106.645,A -85,B 0,C 180,E1 20953.921,E2 20953.921} C_VEL
LIN {X 0,Y 434.51,Z 1099.315,A -85,B 0,C 180,E1 20950.647,E2 20950.647} C_VEL
LIN {X 0,Y 436.175,Z 1091.613,A -85,B 0,C 180,E1 20947.84,E2 20947.84} C_VEL
LIN {X 0,Y 438.816,Z 1080.986,A -85,B 0,C 180,E1 20944.635,E2 20944.635} C_VEL
LIN {X 0,Y 441.682,Z 1070.569,A -85,B 0,C 180,E1 20941.994,E2 20941.994} C_VEL
LIN {X 0,Y 445.622,Z 1057.161,A -85,B 0,C 180,E1 20939.08,E2 20939.08} C_VEL
LIN {X 0,Y 449.559,Z 1044.148,A -85,B 0,C 180,E1 20936.676,E2 20936.676} C_VEL
LIN {X 0,Y 454.394,Z 1028.604,A -85,B 0,C 180,E1 20934.173,E2 20934.173} C_VEL
LIN {X 0,Y 459.409,Z 1011.961,A -85,B 0,C 180,E1 20931.902,E2 20931.902} C_VEL
LIN {X 0,Y 464.735,Z 994.217,A -85,B 0,C 180,E1 20929.8,E2 20929.8} C_VEL
LIN {X 0,Y 469.992,Z 975.534,A -85,B 0,C 180,E1 20927.921,E2 20927.921} C_VEL
LIN {X 0,Y 474.714,Z 957.869,A -85,B 0,C 180,E1 20926.38,E2 20926.38} C_VEL
LIN {X 0,Y 480.116,Z 935.834,A -85,B 0,C 180,E1 20924.743,E2 20924.743} C_VEL
LIN {X 0,Y 484.306,Z 916.935,A -85,B 0,C 180,E1 20923.558,E2 20923.558} C_VEL
LIN {X 0,Y 488.717,Z 894.906,A -85,B 0,C 180,E1 20922.388,E2 20922.388} C_VEL
LIN {X 0,Y 492.369,Z 872.889,A -85,B 0,C 180,E1 20921.44,E2 20921.44} C_VEL
LIN {X 0,Y 495.273,Z 852.424,A -85,B 0,C 180,E1 20920.72,E2 20920.72} C_VEL
LIN {X 0,Y 498.067,Z 827.1,A -85,B 0,C 180,E1 20920.037,E2 20920.037} C_VEL
LIN {X 0,Y 499.696,Z 805.526,A -85,B 0,C 180,E1 20919.611,E2 20919.611} C_VEL
LIN {X 0,Y 511.755,Z 556.719,A -85,B 0,C 180,E1 20915.782,E2 20915.782} C_VEL
LIN {X 0,Y 512.55,Z 538.879,A -85,B 0,C 180,E1 20915.494,E2 20915.494} C_VEL
LIN {X 0,Y 500.945,Z 521.144,A -85,B 0,C 180,E1 20913.258,E2 20913.258} C_VEL
LIN {X 0,Y 490.099,Z 505.859,A -85,B 0,C 180,E1 20910.973,E2 20910.973} C_VEL
LIN {X 0,Y 479.119,Z 491.261,A -85,B 0,C 180,E1 20908.413,E2 20908.413} C_VEL
LIN {X 0,Y 474.276,Z 485.262,A -85,B 0,C 180,E1 20907.191,E2 20907.191} C_VEL
LIN {X 0,Y 470.653,Z 480.698,A -85,B 0,C 180,E1 20906.225,E2 20906.225} C_VEL
LIN {X 0,Y 466.253,Z 475.332,A -85,B 0,C 180,E1 20904.991,E2 20904.991} C_VEL
LIN {X 0,Y 462.52,Z 470.733,A -85,B 0,C 180,E1 20903.879,E2 20903.879} C_VEL
LIN {X 0,Y 458.006,Z 465.617,A -85,B 0,C 180,E1 20902.461,E2 20902.461} C_VEL
LIN {X 0,Y 456.797,Z 463.917,A -85,B 0,C 180,E1 20902.049,E2 20902.049} C_VEL
LIN {X 0,Y 453.391,Z 460.606,A -85,B 0,C 180,E1 20900.899,E2 20900.899} C_VEL
LIN {X 0,Y 451.57,Z 457.774,A -85,B 0,C 180,E1 20900.208,E2 20900.208} C_VEL
LIN {X 0,Y 448.305,Z 455.064,A -85,B 0,C 180,E1 20899.004,E2 20899.004} C_VEL
LIN {X 0,Y 446.323,Z 451.581,A -85,B 0,C 180,E1 20898.144,E2 20898.144} C_VEL
LIN {X 0,Y 443.031,Z 449.405,A -85,B 0,C 180,E1 20896.791,E2 20896.791} C_VEL
LIN {X 0,Y 440.861,Z 446.015,A -85,B 0,C 180,E1 20895.726,E2 20895.726} C_VEL
LIN {X 0,Y 439.987,Z 444.827,A -85,B 0,C 180,E1 20895.285,E2 20895.285} C_VEL
LIN {X 0,Y 436.344,Z 442.453,A -85,B 0,C 180,E1 20893.45,E2 20893.45} C_VEL
LIN {X 0,Y 434.517,Z 438.795,A -85,B 0,C 180,E1 20892.088,E2 20892.088} C_VEL
LIN {X 0,Y 434.403,Z 438.096,A -85,B 0,C 180,E1 20890.88,E2 20890.88} C_VEL
LIN {X 0,Y 434.384,Z 438.082,A -85,B 0,C 180,E1 20887.14,E2 20887.14} C_VEL
LIN {X 0,Y 434.387,Z 438.095,A -85,B 0,C 180,E1 20883.431,E2 20883.431} C_VEL
LIN {X 0,Y 434.398,Z 438.117,A -85,B 0,C 180,E1 20879.604,E2 20879.604} C_VEL
LIN {X 0,Y 434.405,Z 438.088,A -85,B 0,C 180,E1 20875.776,E2 20875.776} C_VEL
LIN {X 0,Y 434.415,Z 438.074,A -85,B 0,C 180,E1 20872.062,E2 20872.062} C_VEL
LIN {X 0,Y 434.411,Z 438.08,A -85,B 0,C 180,E1 20868.314,E2 20868.314} C_VEL
LIN {X 0,Y 434.461,Z 438.392,A -85,B 0,C 180,E1 20865.608,E2 20865.608} C_VEL
LIN {X 0,Y 434.802,Z 439.781,A -85,B 0,C 180,E1 20865,E2 20865} C_VEL
LIN {X 0,Y 436.652,Z 442.71,A -85,B 0,C 180,E1 20863.846,E2 20863.846} C_VEL
LIN {X 0,Y 440.592,Z 445.395,A -85,B 0,C 180,E1 20861.886,E2 20861.886} C_VEL
LIN {X 0,Y 442.578,Z 448.899,A -85,B 0,C 180,E1 20860.877,E2 20860.877} C_VEL
LIN {X 0,Y 446.155,Z 452.01,A -85,B 0,C 180,E1 20859.365,E2 20859.365} C_VEL
LIN {X 0,Y 449.869,Z 456.616,A -85,B 0,C 180,E1 20857.868,E2 20857.868} C_VEL
LIN {X 0,Y 455.126,Z 463.046,A -85,B 0,C 180,E1 20855.95,E2 20855.95} C_VEL
LIN {X 0,Y 458.987,Z 467.861,A -85,B 0,C 180,E1 20854.655,E2 20854.655} C_VEL
LIN {X 0,Y 467.732,Z 479.571,A -85,B 0,C 180,E1 20851.981,E2 20851.981} C_VEL
LIN {X 0,Y 472.569,Z 486.21,A -85,B 0,C 180,E1 20850.636,E2 20850.636} C_VEL
LIN {X 0,Y 478.164,Z 493.937,A -85,B 0,C 180,E1 20849.181,E2 20849.181} C_VEL
LIN {X 0,Y 488.773,Z 509.395,A -85,B 0,C 180,E1 20846.647,E2 20846.647} C_VEL
LIN {X 0,Y 499.742,Z 526.85,A -85,B 0,C 180,E1 20844.268,E2 20844.268} C_VEL
LIN {X 0,Y 510.54,Z 545.315,A -85,B 0,C 180,E1 20842.121,E2 20842.121} C_VEL
LIN {X 0,Y 512.388,Z 548.952,A -85,B 0,C 180,E1 20841.763,E2 20841.763} C_VEL
LIN {X 0,Y 501.921,Z 767.06,A -85,B 0,C 180,E1 20838.405,E2 20838.405} C_VEL
LIN {X 0,Y 498.478,Z 837.007,A -85,B 0,C 180,E1 20837.306,E2 20837.306} C_VEL
LIN {X 0,Y 496.017,Z 862.263,A -85,B 0,C 180,E1 20836.756,E2 20836.756} C_VEL
LIN {X 0,Y 493.232,Z 883.344,A -85,B 0,C 180,E1 20836.152,E2 20836.152} C_VEL
LIN {X 0,Y 489.287,Z 907.858,A -85,B 0,C 180,E1 20835.247,E2 20835.247} C_VEL
LIN {X 0,Y 485.378,Z 928.462,A -85,B 0,C 180,E1 20834.295,E2 20834.295} C_VEL
LIN {X 0,Y 480.583,Z 951.167,A -85,B 0,C 180,E1 20833.034,E2 20833.034} C_VEL
LIN {X 0,Y 475.787,Z 971.177,A -85,B 0,C 180,E1 20831.693,E2 20831.693} C_VEL
LIN {X 0,Y 470.925,Z 990.313,A -85,B 0,C 180,E1 20830.201,E2 20830.201} C_VEL
LIN {X 0,Y 465.418,Z 1010.453,A -85,B 0,C 180,E1 20828.357,E2 20828.357} C_VEL
LIN {X 0,Y 460.598,Z 1027.341,A -85,B 0,C 180,E1 20826.561,E2 20826.561} C_VEL
LIN {X 0,Y 455.317,Z 1045.474,A -85,B 0,C 180,E1 20824.339,E2 20824.339} C_VEL
LIN {X 0,Y 450.568,Z 1061.553,A -85,B 0,C 180,E1 20822.032,E2 20822.032} C_VEL
LIN {X 0,Y 445.998,Z 1077.457,A -85,B 0,C 180,E1 20819.405,E2 20819.405} C_VEL
LIN {X 0,Y 442.12,Z 1091.322,A -85,B 0,C 180,E1 20816.705,E2 20816.705} C_VEL
LIN {X 0,Y 438.796,Z 1104.309,A -85,B 0,C 180,E1 20813.787,E2 20813.787} C_VEL
LIN {X 0,Y 436.211,Z 1115.374,A -85,B 0,C 180,E1 20810.812,E2 20810.812} C_VEL
LIN {X 0,Y 434.365,Z 1124.86,A -85,B 0,C 180,E1 20807.828,E2 20807.828} C_VEL
LIN {X 0,Y 433.071,Z 1133.001,A -85,B 0,C 180,E1 20804.668,E2 20804.668} C_VEL
LIN {X 0,Y 432.428,Z 1138.599,A -85,B 0,C 180,E1 20802.011,E2 20802.011} C_VEL
LIN {X 0,Y 432.059,Z 1143.915,A -85,B 0,C 180,E1 20798.786,E2 20798.786} C_VEL
LIN {X 0,Y 431.965,Z 1147.203,A -85,B 0,C 180,E1 20795.846,E2 20795.846} C_VEL
LIN {X 0,Y 431.957,Z 1149.061,A -85,B 0,C 180,E1 20793.185,E2 20793.185} C_VEL
LIN {X 0,Y 431.98,Z 1149.887,A -85,B 0,C 180,E1 20790.133,E2 20790.133} C_VEL
LIN {X 0,Y 431.957,Z 1149.133,A -85,B 0,C 180,E1 20787.214,E2 20787.214} C_VEL
LIN {X 0,Y 431.951,Z 1147.437,A -85,B 0,C 180,E1 20784.687,E2 20784.687} C_VEL
LIN {X 0,Y 432.009,Z 1144.562,A -85,B 0,C 180,E1 20782.017,E2 20782.017} C_VEL
LIN {X 0,Y 432.31,Z 1139.421,A -85,B 0,C 180,E1 20778.717,E2 20778.717} C_VEL
LIN {X 0,Y 432.874,Z 1133.704,A -85,B 0,C 180,E1 20775.964,E2 20775.964} C_VEL
LIN {X 0,Y 433.925,Z 1126.146,A -85,B 0,C 180,E1 20772.984,E2 20772.984} C_VEL
LIN {X 0,Y 435.65,Z 1116.298,A -85,B 0,C 180,E1 20769.839,E2 20769.839} C_VEL
LIN {X 0,Y 437.747,Z 1106.359,A -85,B 0,C 180,E1 20767.15,E2 20767.15} C_VEL
LIN {X 0,Y 440.942,Z 1092.812,A -85,B 0,C 180,E1 20764.046,E2 20764.046} C_VEL
LIN {X 0,Y 444.256,Z 1079.826,A -85,B 0,C 180,E1 20761.5,E2 20761.5} C_VEL
LIN {X 0,Y 448.707,Z 1063.282,A -85,B 0,C 180,E1 20758.72,E2 20758.72} C_VEL
LIN {X 0,Y 452.675,Z 1048.744,A -85,B 0,C 180,E1 20756.61,E2 20756.61} C_VEL
LIN {X 0,Y 457.658,Z 1030.564,A -85,B 0,C 180,E1 20754.314,E2 20754.314} C_VEL
LIN {X 0,Y 462.327,Z 1013.013,A -85,B 0,C 180,E1 20752.418,E2 20752.418} C_VEL
LIN {X 0,Y 467.547,Z 992.943,A -85,B 0,C 180,E1 20750.537,E2 20750.537} C_VEL
LIN {X 0,Y 472.467,Z 972.331,A -85,B 0,C 180,E1 20748.911,E2 20748.911} C_VEL
LIN {X 0,Y 476.999,Z 952.197,A -85,B 0,C 180,E1 20747.547,E2 20747.547} C_VEL
LIN {X 0,Y 481.581,Z 929.283,A -85,B 0,C 180,E1 20746.259,E2 20746.259} C_VEL
LIN {X 0,Y 485.083,Z 909.703,A -85,B 0,C 180,E1 20745.34,E2 20745.34} C_VEL
LIN {X 0,Y 488.904,Z 884.901,A -85,B 0,C 180,E1 20744.399,E2 20744.399} C_VEL
LIN {X 0,Y 491.565,Z 863.698,A -85,B 0,C 180,E1 20743.776,E2 20743.776} C_VEL
LIN {X 0,Y 493.903,Z 839.183,A -85,B 0,C 180,E1 20743.224,E2 20743.224} C_VEL
LIN {X 0,Y 496.447,Z 785.173,A -85,B 0,C 180,E1 20742.368,E2 20742.368} C_VEL
LIN {X 0,Y 506.053,Z 566.692,A -85,B 0,C 180,E1 20739.015,E2 20739.015} C_VEL
LIN {X 0,Y 506.86,Z 545.654,A -85,B 0,C 180,E1 20738.672,E2 20738.672} C_VEL
LIN {X 0,Y 495.661,Z 525.648,A -85,B 0,C 180,E1 20736.664,E2 20736.664} C_VEL
LIN {X 0,Y 484.104,Z 506.731,A -85,B 0,C 180,E1 20734.431,E2 20734.431} C_VEL
LIN {X 0,Y 472.248,Z 488.773,A -85,B 0,C 180,E1 20731.924,E2 20731.924} C_VEL
LIN {X 0,Y 462.563,Z 475.097,A -85,B 0,C 180,E1 20729.671,E2 20729.671} C_VEL
LIN {X 0,Y 454.842,Z 464.763,A -85,B 0,C 180,E1 20727.707,E2 20727.707} C_VEL
LIN {X 0,Y 451.257,Z 460.041,A -85,B 0,C 180,E1 20726.731,E2 20726.731} C_VEL
LIN {X 0,Y 446.879,Z 454.382,A -85,B 0,C 180,E1 20725.478,E2 20725.478} C_VEL
LIN {X 0,Y 442.658,Z 449.262,A -85,B 0,C 180,E1 20724.204,E2 20724.204} C_VEL
LIN {X 0,Y 438.553,Z 444.183,A -85,B 0,C 180,E1 20722.876,E2 20722.876} C_VEL
LIN {X 0,Y 435.695,Z 441.567,A -85,B 0,C 180,E1 20721.932,E2 20721.932} C_VEL
LIN {X 0,Y 434.518,Z 438.712,A -85,B 0,C 180,E1 20721.32,E2 20721.32} C_VEL
LIN {X 0,Y 434.416,Z 438.106,A -85,B 0,C 180,E1 20720.619,E2 20720.619} C_VEL
LIN {X 0,Y 434.412,Z 438.118,A -85,B 0,C 180,E1 20716.761,E2 20716.761} C_VEL
LIN {X 0,Y 434.404,Z 438.082,A -85,B 0,C 180,E1 20712.901,E2 20712.901} C_VEL
LIN {X 0,Y 434.403,Z 438.07,A -85,B 0,C 180,E1 20709.139,E2 20709.139} C_VEL
LIN {X 0,Y 434.416,Z 438.109,A -85,B 0,C 180,E1 20705.415,E2 20705.415} C_VEL
LIN {X 0,Y 434.417,Z 438.086,A -85,B 0,C 180,E1 20701.583,E2 20701.583} C_VEL
LIN {X 0,Y 434.41,Z 438.068,A -85,B 0,C 180,E1 20697.889,E2 20697.889} C_VEL
LIN {X 0,Y 434.404,Z 438.107,A -85,B 0,C 180,E1 20694.055,E2 20694.055} C_VEL
LIN {X 0,Y 434.383,Z 438.089,A -85,B 0,C 180,E1 20690.326,E2 20690.326} C_VEL
LIN {X 0,Y 434.374,Z 438.073,A -85,B 0,C 180,E1 20686.556,E2 20686.556} C_VEL
LIN {X 0,Y 434.391,Z 438.101,A -85,B 0,C 180,E1 20682.864,E2 20682.864} C_VEL
LIN {X 0,Y 434.407,Z 438.101,A -85,B 0,C 180,E1 20679.098,E2 20679.098} C_VEL
LIN {X 0,Y 434.419,Z 438.17,A -85,B 0,C 180,E1 20675.38,E2 20675.38} C_VEL
LIN {X 0,Y 434.7,Z 439.504,A -85,B 0,C 180,E1 20674.93,E2 20674.93} C_VEL
LIN {X 0,Y 436.347,Z 442.457,A -85,B 0,C 180,E1 20674.299,E2 20674.299} C_VEL
LIN {X 0,Y 439.31,Z 444.535,A -85,B 0,C 180,E1 20673.36,E2 20673.36} C_VEL
LIN {X 0,Y 439.969,Z 445.24,A -85,B 0,C 180,E1 20673.148,E2 20673.148} C_VEL
LIN {X 0,Y 442.148,Z 448.8,A -85,B 0,C 180,E1 20672.417,E2 20672.417} C_VEL
LIN {X 0,Y 445.279,Z 451.45,A -85,B 0,C 180,E1 20671.499,E2 20671.499} C_VEL
LIN {X 0,Y 448.035,Z 455.427,A -85,B 0,C 180,E1 20670.668,E2 20670.668} C_VEL
LIN {X 0,Y 450.475,Z 457.684,A -85,B 0,C 180,E1 20670.002,E2 20670.002} C_VEL
LIN {X 0,Y 453.731,Z 461.951,A -85,B 0,C 180,E1 20669.105,E2 20669.105} C_VEL
LIN {X 0,Y 455.686,Z 464.047,A -85,B 0,C 180,E1 20668.599,E2 20668.599} C_VEL
LIN {X 0,Y 459.485,Z 468.589,A -85,B 0,C 180,E1 20667.634,E2 20667.634} C_VEL
LIN {X 0,Y 469.578,Z 481.561,A -85,B 0,C 180,E1 20665.24,E2 20665.24} C_VEL
LIN {X 0,Y 480.587,Z 496.06,A -85,B 0,C 180,E1 20662.889,E2 20662.889} C_VEL
LIN {X 0,Y 491.103,Z 511.074,A -85,B 0,C 180,E1 20660.826,E2 20660.826} C_VEL
LIN {X 0,Y 503.524,Z 529.946,A -85,B 0,C 180,E1 20658.584,E2 20658.584} C_VEL
LIN {X 0,Y 507.263,Z 536.253,A -85,B 0,C 180,E1 20657.937,E2 20657.937} C_VEL
LIN {X 0,Y 496.222,Z 782.654,A -85,B 0,C 180,E1 20654.17,E2 20654.17} C_VEL
LIN {X 0,Y 494.378,Z 817.794,A -85,B 0,C 180,E1 20653.585,E2 20653.585} C_VEL
LIN {X 0,Y 492.281,Z 840.5,A -85,B 0,C 180,E1 20653.042,E2 20653.042} C_VEL
LIN {X 0,Y 489.434,Z 864.549,A -85,B 0,C 180,E1 20652.286,E2 20652.286} C_VEL
LIN {X 0,Y 486.088,Z 886.593,A -85,B 0,C 180,E1 20651.388,E2 20651.388} C_VEL
LIN {X 0,Y 482.391,Z 907.908,A -85,B 0,C 180,E1 20650.34,E2 20650.34} C_VEL
LIN {X 0,Y 477.935,Z 929.939,A -85,B 0,C 180,E1 20649.03,E2 20649.03} C_VEL
LIN {X 0,Y 473.823,Z 948.422,A -85,B 0,C 180,E1 20647.733,E2 20647.733} C_VEL
LIN {X 0,Y 468.706,Z 969.601,A -85,B 0,C 180,E1 20645.996,E2 20645.996} C_VEL
LIN {X 0,Y 464.077,Z 987.281,A -85,B 0,C 180,E1 20644.293,E2 20644.293} C_VEL
LIN {X 0,Y 459.072,Z 1005.734,A -85,B 0,C 180,E1 20642.251,E2 20642.251} C_VEL
LIN {X 0,Y 454.108,Z 1023.047,A -85,B 0,C 180,E1 20639.989,E2 20639.989} C_VEL
LIN {X 0,Y 449.544,Z 1039.199,A -85,B 0,C 180,E1 20637.558,E2 20637.558} C_VEL
LIN {X 0,Y 445.345,Z 1053.784,A -85,B 0,C 180,E1 20634.967,E2 20634.967} C_VEL
LIN {X 0,Y 441.692,Z 1067.297,A -85,B 0,C 180,E1 20632.197,E2 20632.197} C_VEL
LIN {X 0,Y 438.57,Z 1079.178,A -85,B 0,C 180,E1 20629.286,E2 20629.286} C_VEL
LIN {X 0,Y 436.22,Z 1089.352,A -85,B 0,C 180,E1 20626.376,E2 20626.376} C_VEL
LIN {X 0,Y 434.417,Z 1098.117,A -85,B 0,C 180,E1 20623.307,E2 20623.307} C_VEL
LIN {X 0,Y 433.302,Z 1104.751,A -85,B 0,C 180,E1 20620.504,E2 20620.504} C_VEL
LIN {X 0,Y 432.536,Z 1110.717,A -85,B 0,C 180,E1 20617.302,E2 20617.302} C_VEL
LIN {X 0,Y 431.4,Z 1112.294,A -85,B 0,C 180,E1 20616.304,E2 20616.304} C_VEL
LIN {X 0,Y 426.747,Z 1114.894,A -85,B 0,C 180,E1 20614.494,E2 20614.494} C_VEL
LIN {X 0,Y 424.315,Z 1116.386,A -85,B 0,C 180,E1 20613.192,E2 20613.192} C_VEL
LIN {X 0,Y 424.092,Z 1116.75,A -85,B 0,C 180,E1 20612.744,E2 20612.744} C_VEL
LIN {X 0,Y 424.017,Z 1118.646,A -85,B 0,C 180,E1 20609.865,E2 20609.865} C_VEL
LIN {X 0,Y 423.982,Z 1119.409,A -85,B 0,C 180,E1 20606.62,E2 20606.62} C_VEL
LIN {X 0,Y 424.029,Z 1118.642,A -85,B 0,C 180,E1 20603.637,E2 20603.637} C_VEL
LIN {X 0,Y 424.12,Z 1116.881,A -85,B 0,C 180,E1 20600.912,E2 20600.912} C_VEL
LIN {X 0,Y 424.427,Z 1113.385,A -85,B 0,C 180,E1 20597.621,E2 20597.621} C_VEL
LIN {X 0,Y 425.056,Z 1108.612,A -85,B 0,C 180,E1 20594.584,E2 20594.584} C_VEL
LIN {X 0,Y 426.082,Z 1102.8,A -85,B 0,C 180,E1 20591.672,E2 20591.672} C_VEL
LIN {X 0,Y 427.893,Z 1094.412,A -85,B 0,C 180,E1 20588.333,E2 20588.333} C_VEL
LIN {X 0,Y 430.006,Z 1085.92,A -85,B 0,C 180,E1 20585.55,E2 20585.55} C_VEL
LIN {X 0,Y 433.261,Z 1074.365,A -85,B 0,C 180,E1 20582.363,E2 20582.363} C_VEL
LIN {X 0,Y 436.853,Z 1062.477,A -85,B 0,C 180,E1 20579.613,E2 20579.613} C_VEL
LIN {X 0,Y 441.188,Z 1048.847,A -85,B 0,C 180,E1 20576.894,E2 20576.894} C_VEL
LIN {X 0,Y 445.721,Z 1034.591,A -85,B 0,C 180,E1 20574.478,E2 20574.478} C_VEL
LIN {X 0,Y 450.811,Z 1018.818,A -85,B 0,C 180,E1 20572.149,E2 20572.149} C_VEL
LIN {X 0,Y 456.36,Z 1000.891,A -85,B 0,C 180,E1 20569.897,E2 20569.897} C_VEL
LIN {X 0,Y 461.47,Z 983.91,A -85,B 0,C 180,E1 20568.053,E2 20568.053} C_VEL
LIN {X 0,Y 467.376,Z 962.989,A -85,B 0,C 180,E1 20566.119,E2 20566.119} C_VEL
LIN {X 0,Y 472.249,Z 944.352,A -85,B 0,C 180,E1 20564.65,E2 20564.65} C_VEL
LIN {X 0,Y 477.602,Z 921.778,A -85,B 0,C 180,E1 20563.146,E2 20563.146} C_VEL
LIN {X 0,Y 481.662,Z 902.512,A -85,B 0,C 180,E1 20562.074,E2 20562.074} C_VEL
LIN {X 0,Y 485.845,Z 879.985,A -85,B 0,C 180,E1 20561.017,E2 20561.017} C_VEL
LIN {X 0,Y 489.285,Z 857.026,A -85,B 0,C 180,E1 20560.168,E2 20560.168} C_VEL
LIN {X 0,Y 492.162,Z 833.74,A -85,B 0,C 180,E1 20559.489,E2 20559.489} C_VEL
LIN {X 0,Y 494.223,Z 809.258,A -85,B 0,C 180,E1 20558.975,E2 20558.975} C_VEL
LIN {X 0,Y 505.833,Z 578.003,A -85,B 0,C 180,E1 20555.388,E2 20555.388} C_VEL
LIN {X 0,Y 507.595,Z 542.865,A -85,B 0,C 180,E1 20554.838,E2 20554.838} C_VEL
LIN {X 0,Y 496.248,Z 525.655,A -85,B 0,C 180,E1 20552.581,E2 20552.581} C_VEL
LIN {X 0,Y 487.008,Z 512.42,A -85,B 0,C 180,E1 20550.575,E2 20550.575} C_VEL
LIN {X 0,Y 476.177,Z 497.879,A -85,B 0,C 180,E1 20547.99,E2 20547.99} C_VEL
LIN {X 0,Y 468.457,Z 488.051,A -85,B 0,C 180,E1 20545.948,E2 20545.948} C_VEL
LIN {X 0,Y 463.71,Z 482.308,A -85,B 0,C 180,E1 20544.593,E2 20544.593} C_VEL
LIN {X 0,Y 459.203,Z 476.792,A -85,B 0,C 180,E1 20543.211,E2 20543.211} C_VEL
LIN {X 0,Y 455.539,Z 472.349,A -85,B 0,C 180,E1 20542.011,E2 20542.011} C_VEL
LIN {X 0,Y 454.047,Z 470.796,A -85,B 0,C 180,E1 20541.51,E2 20541.51} C_VEL
LIN {X 0,Y 450.703,Z 466.893,A -85,B 0,C 180,E1 20540.316,E2 20540.316} C_VEL
LIN {X 0,Y 449.609,Z 465.279,A -85,B 0,C 180,E1 20539.893,E2 20539.893} C_VEL
LIN {X 0,Y 446.265,Z 462.224,A -85,B 0,C 180,E1 20538.62,E2 20538.62} C_VEL
LIN {X 0,Y 444.443,Z 459.178,A -85,B 0,C 180,E1 20537.817,E2 20537.817} C_VEL
LIN {X 0,Y 441.102,Z 456.639,A -85,B 0,C 180,E1 20536.393,E2 20536.393} C_VEL
LIN {X 0,Y 438.767,Z 452.715,A -85,B 0,C 180,E1 20535.193,E2 20535.193} C_VEL
LIN {X 0,Y 435.03,Z 450.262,A -85,B 0,C 180,E1 20533.288,E2 20533.288} C_VEL
LIN {X 0,Y 433.129,Z 446.951,A -85,B 0,C 180,E1 20532.059,E2 20532.059} C_VEL
LIN {X 0,Y 432.029,Z 445.797,A -85,B 0,C 180,E1 20531.346,E2 20531.346} C_VEL
LIN {X 0,Y 428.537,Z 443.551,A -85,B 0,C 180,E1 20528.859,E2 20528.859} C_VEL
LIN {X 0,Y 426.727,Z 440.373,A -85,B 0,C 180,E1 20526.999,E2 20526.999} C_VEL
LIN {X 0,Y 426.475,Z 439.241,A -85,B 0,C 180,E1 20525.786,E2 20525.786} C_VEL
LIN {X 0,Y 426.467,Z 439.062,A -85,B 0,C 180,E1 20522.015,E2 20522.015} C_VEL
LIN {X 0,Y 426.477,Z 439.067,A -85,B 0,C 180,E1 20518.253,E2 20518.253} C_VEL
LIN {X 0,Y 426.48,Z 439.088,A -85,B 0,C 180,E1 20514.349,E2 20514.349} C_VEL
LIN {X 0,Y 426.504,Z 439.376,A -85,B 0,C 180,E1 20511.371,E2 20511.371} C_VEL
LIN {X 0,Y 426.807,Z 440.577,A -85,B 0,C 180,E1 20510.357,E2 20510.357} C_VEL
LIN {X 0,Y 428.593,Z 443.574,A -85,B 0,C 180,E1 20508.562,E2 20508.562} C_VEL
LIN {X 0,Y 432.966,Z 446.552,A -85,B 0,C 180,E1 20505.523,E2 20505.523} C_VEL
LIN {X 0,Y 434.785,Z 449.909,A -85,B 0,C 180,E1 20504.323,E2 20504.323} C_VEL
LIN {X 0,Y 438.063,Z 452.399,A -85,B 0,C 180,E1 20502.602,E2 20502.602} C_VEL
LIN {X 0,Y 438.969,Z 453.108,A -85,B 0,C 180,E1 20502.16,E2 20502.16} C_VEL
LIN {X 0,Y 441.206,Z 456.756,A -85,B 0,C 180,E1 20501.022,E2 20501.022} C_VEL
LIN {X 0,Y 444.524,Z 459.68,A -85,B 0,C 180,E1 20499.595,E2 20499.595} C_VEL
LIN {X 0,Y 448.117,Z 464.167,A -85,B 0,C 180,E1 20498.122,E2 20498.122} C_VEL
LIN {X 0,Y 453.13,Z 470.47,A -85,B 0,C 180,E1 20496.252,E2 20496.252} C_VEL
LIN {X 0,Y 458.172,Z 477.05,A -85,B 0,C 180,E1 20494.537,E2 20494.537} C_VEL
LIN {X 0,Y 465.282,Z 486.602,A -85,B 0,C 180,E1 20492.342,E2 20492.342} C_VEL
LIN {X 0,Y 472.947,Z 497.154,A -85,B 0,C 180,E1 20490.209,E2 20490.209} C_VEL
LIN {X 0,Y 482.208,Z 510.775,A -85,B 0,C 180,E1 20487.868,E2 20487.868} C_VEL
LIN {X 0,Y 492.139,Z 526.169,A -85,B 0,C 180,E1 20485.591,E2 20485.591} C_VEL
LIN {X 0,Y 502.764,Z 544.153,A -85,B 0,C 180,E1 20483.353,E2 20483.353} C_VEL
LIN {X 0,Y 507.388,Z 552.709,A -85,B 0,C 180,E1 20482.427,E2 20482.427} C_VEL
LIN {X 0,Y 496.568,Z 770.754,A -85,B 0,C 180,E1 20479.051,E2 20479.051} C_VEL
LIN {X 0,Y 493.179,Z 837.021,A -85,B 0,C 180,E1 20478.001,E2 20478.001} C_VEL
LIN {X 0,Y 490.665,Z 862.01,A -85,B 0,C 180,E1 20477.454,E2 20477.454} C_VEL
LIN {X 0,Y 487.761,Z 883.379,A -85,B 0,C 180,E1 20476.84,E2 20476.84} C_VEL
LIN {X 0,Y 483.659,Z 908.033,A -85,B 0,C 180,E1 20475.923,E2 20475.923} C_VEL
LIN {X 0,Y 479.636,Z 928.582,A -85,B 0,C 180,E1 20474.968,E2 20474.968} C_VEL
LIN {X 0,Y 474.692,Z 951.201,A -85,B 0,C 180,E1 20473.702,E2 20473.702} C_VEL
LIN {X 0,Y 469.742,Z 971.176,A -85,B 0,C 180,E1 20472.354,E2 20472.354} C_VEL
LIN {X 0,Y 464.527,Z 991.02,A -85,B 0,C 180,E1 20470.79,E2 20470.79} C_VEL
LIN {X 0,Y 458.709,Z 1011.413,A -85,B 0,C 180,E1 20468.887,E2 20468.887} C_VEL
LIN {X 0,Y 453.805,Z 1027.97,A -85,B 0,C 180,E1 20467.097,E2 20467.097} C_VEL
LIN {X 0,Y 447.971,Z 1047.082,A -85,B 0,C 180,E1 20464.693,E2 20464.693} C_VEL
LIN {X 0,Y 443.314,Z 1062.257,A -85,B 0,C 180,E1 20462.467,E2 20462.467} C_VEL
LIN {X 0,Y 438.302,Z 1078.862,A -85,B 0,C 180,E1 20459.637,E2 20459.637} C_VEL
LIN {X 0,Y 434.556,Z 1091.745,A -85,B 0,C 180,E1 20457.067,E2 20457.067} C_VEL
LIN {X 0,Y 431.085,Z 1104.623,A -85,B 0,C 180,E1 20454.094,E2 20454.094} C_VEL
LIN {X 0,Y 428.501,Z 1115.156,A -85,B 0,C 180,E1 20451.204,E2 20451.204} C_VEL
LIN {X 0,Y 426.467,Z 1125.037,A -85,B 0,C 180,E1 20448.028,E2 20448.028} C_VEL
LIN {X 0,Y 425.12,Z 1133.019,A -85,B 0,C 180,E1 20444.831,E2 20444.831} C_VEL
LIN {X 0,Y 424.418,Z 1138.87,A -85,B 0,C 180,E1 20441.965,E2 20441.965} C_VEL
LIN {X 0,Y 424.053,Z 1144.146,A -85,B 0,C 180,E1 20438.543,E2 20438.543} C_VEL
LIN {X 0,Y 423.965,Z 1147.051,A -85,B 0,C 180,E1 20435.821,E2 20435.821} C_VEL
LIN {X 0,Y 423.959,Z 1148.856,A -85,B 0,C 180,E1 20433.11,E2 20433.11} C_VEL
LIN {X 0,Y 423.994,Z 1149.581,A -85,B 0,C 180,E1 20430,E2 20430} C_VEL
LIN {X 0,Y 423.961,Z 1148.768,A -85,B 0,C 180,E1 20427.026,E2 20427.026} C_VEL
LIN {X 0,Y 423.959,Z 1146.997,A -85,B 0,C 180,E1 20424.428,E2 20424.428} C_VEL
LIN {X 0,Y 424.056,Z 1143.757,A -85,B 0,C 180,E1 20421.457,E2 20421.457} C_VEL
LIN {X 0,Y 424.385,Z 1138.461,A -85,B 0,C 180,E1 20418.172,E2 20418.172} C_VEL
LIN {X 0,Y 425.015,Z 1132.741,A -85,B 0,C 180,E1 20415.42,E2 20415.42} C_VEL
LIN {X 0,Y 426.26,Z 1124.641,A -85,B 0,C 180,E1 20412.245,E2 20412.245} C_VEL
LIN {X 0,Y 427.975,Z 1115.535,A -85,B 0,C 180,E1 20409.342,E2 20409.342} C_VEL
LIN {X 0,Y 430.365,Z 1104.922,A -85,B 0,C 180,E1 20406.446,E2 20406.446} C_VEL
LIN {X 0,Y 433.642,Z 1091.758,A -85,B 0,C 180,E1 20403.428,E2 20403.428} C_VEL
LIN {X 0,Y 437.159,Z 1078.693,A -85,B 0,C 180,E1 20400.844,E2 20400.844} C_VEL
LIN {X 0,Y 441.747,Z 1062.343,A -85,B 0,C 180,E1 20398.083,E2 20398.083} C_VEL
LIN {X 0,Y 446.257,Z 1046.534,A -85,B 0,C 180,E1 20395.778,E2 20395.778} C_VEL
LIN {X 0,Y 451.563,Z 1027.812,A -85,B 0,C 180,E1 20393.441,E2 20393.441} C_VEL
LIN {X 0,Y 456.316,Z 1010.646,A -85,B 0,C 180,E1 20391.595,E2 20391.595} C_VEL
LIN {X 0,Y 461.95,Z 989.347,A -85,B 0,C 180,E1 20389.633,E2 20389.633} C_VEL
LIN {X 0,Y 466.469,Z 971.006,A -85,B 0,C 180,E1 20388.192,E2 20388.192} C_VEL
LIN {X 0,Y 471.406,Z 949.701,A -85,B 0,C 180,E1 20386.756,E2 20386.756} C_VEL
LIN {X 0,Y 475.903,Z 927.53,A -85,B 0,C 180,E1 20385.524,E2 20385.524} C_VEL
LIN {X 0,Y 480.015,Z 905.047,A -85,B 0,C 180,E1 20384.484,E2 20384.484} C_VEL
LIN {X 0,Y 483.627,Z 881.15,A -85,B 0,C 180,E1 20383.618,E2 20383.618} C_VEL
LIN {X 0,Y 486.436,Z 858.827,A -85,B 0,C 180,E1 20382.986,E2 20382.986} C_VEL
LIN {X 0,Y 488.636,Z 833.303,A -85,B 0,C 180,E1 20382.454,E2 20382.454} C_VEL
LIN {X 0,Y 498.879,Z 609.362,A -85,B 0,C 180,E1 20378.978,E2 20378.978} C_VEL
LIN {X 0,Y 501.551,Z 549.09,A -85,B 0,C 180,E1 20378.026,E2 20378.026} C_VEL
LIN {X 0,Y 490.022,Z 528.473,A -85,B 0,C 180,E1 20375.887,E2 20375.887} C_VEL
LIN {X 0,Y 479.538,Z 511.426,A -85,B 0,C 180,E1 20373.794,E2 20373.794} C_VEL
LIN {X 0,Y 469.09,Z 495.324,A -85,B 0,C 180,E1 20371.518,E2 20371.518} C_VEL
LIN {X 0,Y 459.649,Z 481.823,A -85,B 0,C 180,E1 20369.269,E2 20369.269} C_VEL
LIN {X 0,Y 451.724,Z 471.081,A -85,B 0,C 180,E1 20367.199,E2 20367.199} C_VEL
LIN {X 0,Y 448.612,Z 466.941,A -85,B 0,C 180,E1 20366.33,E2 20366.33} C_VEL
LIN {X 0,Y 444.2,Z 461.202,A -85,B 0,C 180,E1 20365.036,E2 20365.036} C_VEL
LIN {X 0,Y 439.865,Z 455.893,A -85,B 0,C 180,E1 20363.69,E2 20363.69} C_VEL
LIN {X 0,Y 436.476,Z 451.609,A -85,B 0,C 180,E1 20362.564,E2 20362.564} C_VEL
LIN {X 0,Y 433.492,Z 448.694,A -85,B 0,C 180,E1 20361.551,E2 20361.551} C_VEL
LIN {X 0,Y 431.785,Z 445.748,A -85,B 0,C 180,E1 20360.893,E2 20360.893} C_VEL
LIN {X 0,Y 428.329,Z 443.276,A -85,B 0,C 180,E1 20359.643,E2 20359.643} C_VEL
LIN {X 0,Y 426.579,Z 439.712,A -85,B 0,C 180,E1 20358.731,E2 20358.731} C_VEL
LIN {X 0,Y 426.474,Z 439.096,A -85,B 0,C 180,E1 20358.028,E2 20358.028} C_VEL
LIN {X 0,Y 426.48,Z 439.057,A -85,B 0,C 180,E1 20354.251,E2 20354.251} C_VEL
LIN {X 0,Y 426.47,Z 439.08,A -85,B 0,C 180,E1 20350.401,E2 20350.401} C_VEL
LIN {X 0,Y 426.463,Z 439.091,A -85,B 0,C 180,E1 20346.597,E2 20346.597} C_VEL
LIN {X 0,Y 426.452,Z 439.058,A -85,B 0,C 180,E1 20342.688,E2 20342.688} C_VEL
LIN {X 0,Y 426.459,Z 439.073,A -85,B 0,C 180,E1 20338.925,E2 20338.925} C_VEL
LIN {X 0,Y 426.468,Z 439.097,A -85,B 0,C 180,E1 20335.158,E2 20335.158} C_VEL
LIN {X 0,Y 426.476,Z 439.055,A -85,B 0,C 180,E1 20331.37,E2 20331.37} C_VEL
LIN {X 0,Y 426.476,Z 439.067,A -85,B 0,C 180,E1 20327.543,E2 20327.543} C_VEL
